(* IEC 61131-3 sources: TA/Tests/RetainTest/OLD/Structure test (part 8) *)

    ARRAY_ARRAY_STRUCTURE_AUTO.ARRAY_ARRAY_SINT[3][0] := ARRAY_ARRAY_STRUCTURE_AUTO.ARRAY_ARRAY_SINT[3][0] + 1;
    ARRAY_ARRAY_STRUCTURE_AUTO.ARRAY_ARRAY_SINT[3][1] := ARRAY_ARRAY_STRUCTURE_AUTO.ARRAY_ARRAY_SINT[3][1] + 1;
    ARRAY_ARRAY_STRUCTURE_AUTO.ARRAY_ARRAY_SINT[3][2] := ARRAY_ARRAY_STRUCTURE_AUTO.ARRAY_ARRAY_SINT[3][2] + 1;
    ARRAY_ARRAY_STRUCTURE_AUTO.ARRAY_ARRAY_SINT[3][3] := ARRAY_ARRAY_STRUCTURE_AUTO.ARRAY_ARRAY_SINT[3][3] + 1;
    ARRAY_ARRAY_STRUCTURE_AUTO.ARRAY_ARRAY_SINT[3][4] := ARRAY_ARRAY_STRUCTURE_AUTO.ARRAY_ARRAY_SINT[3][4] + 1;
    ARRAY_ARRAY_STRUCTURE_AUTO.ARRAY_ARRAY_SINT[3][5] := ARRAY_ARRAY_STRUCTURE_AUTO.ARRAY_ARRAY_SINT[3][5] + 1;
    ARRAY_ARRAY_STRUCTURE_AUTO.ARRAY_ARRAY_SINT[3][6] := ARRAY_ARRAY_STRUCTURE_AUTO.ARRAY_ARRAY_SINT[3][6] + 1;
    ARRAY_ARRAY_STRUCTURE_AUTO.ARRAY_ARRAY_SINT[3][7] := ARRAY_ARRAY_STRUCTURE_AUTO.ARRAY_ARRAY_SINT[3][7] + 1;
    ARRAY_ARRAY_STRUCTURE_AUTO.ARRAY_ARRAY_SINT[3][8] := ARRAY_ARRAY_STRUCTURE_AUTO.ARRAY_ARRAY_SINT[3][8] + 1;
    ARRAY_ARRAY_STRUCTURE_AUTO.ARRAY_ARRAY_SINT[3][9] := ARRAY_ARRAY_STRUCTURE_AUTO.ARRAY_ARRAY_SINT[3][9] + 1;

    ARRAY_ARRAY_STRUCTURE_AUTO.ARRAY_ARRAY_SINT[4][0] := ARRAY_ARRAY_STRUCTURE_AUTO.ARRAY_ARRAY_SINT[4][0] + 1;
    ARRAY_ARRAY_STRUCTURE_AUTO.ARRAY_ARRAY_SINT[4][1] := ARRAY_ARRAY_STRUCTURE_AUTO.ARRAY_ARRAY_SINT[4][1] + 1;
    ARRAY_ARRAY_STRUCTURE_AUTO.ARRAY_ARRAY_SINT[4][2] := ARRAY_ARRAY_STRUCTURE_AUTO.ARRAY_ARRAY_SINT[4][2] + 1;
    ARRAY_ARRAY_STRUCTURE_AUTO.ARRAY_ARRAY_SINT[4][3] := ARRAY_ARRAY_STRUCTURE_AUTO.ARRAY_ARRAY_SINT[4][3] + 1;
    ARRAY_ARRAY_STRUCTURE_AUTO.ARRAY_ARRAY_SINT[4][4] := ARRAY_ARRAY_STRUCTURE_AUTO.ARRAY_ARRAY_SINT[4][4] + 1;
    ARRAY_ARRAY_STRUCTURE_AUTO.ARRAY_ARRAY_SINT[4][5] := ARRAY_ARRAY_STRUCTURE_AUTO.ARRAY_ARRAY_SINT[4][5] + 1;
    ARRAY_ARRAY_STRUCTURE_AUTO.ARRAY_ARRAY_SINT[4][6] := ARRAY_ARRAY_STRUCTURE_AUTO.ARRAY_ARRAY_SINT[4][6] + 1;
    ARRAY_ARRAY_STRUCTURE_AUTO.ARRAY_ARRAY_SINT[4][7] := ARRAY_ARRAY_STRUCTURE_AUTO.ARRAY_ARRAY_SINT[4][7] + 1;
    ARRAY_ARRAY_STRUCTURE_AUTO.ARRAY_ARRAY_SINT[4][8] := ARRAY_ARRAY_STRUCTURE_AUTO.ARRAY_ARRAY_SINT[4][8] + 1;
    ARRAY_ARRAY_STRUCTURE_AUTO.ARRAY_ARRAY_SINT[4][9] := ARRAY_ARRAY_STRUCTURE_AUTO.ARRAY_ARRAY_SINT[4][9] + 1;

    ARRAY_ARRAY_STRUCTURE_AUTO.ARRAY_ARRAY_SINT[5][0] := ARRAY_ARRAY_STRUCTURE_AUTO.ARRAY_ARRAY_SINT[5][0] + 1;
    ARRAY_ARRAY_STRUCTURE_AUTO.ARRAY_ARRAY_SINT[5][1] := ARRAY_ARRAY_STRUCTURE_AUTO.ARRAY_ARRAY_SINT[5][1] + 1;
    ARRAY_ARRAY_STRUCTURE_AUTO.ARRAY_ARRAY_SINT[5][2] := ARRAY_ARRAY_STRUCTURE_AUTO.ARRAY_ARRAY_SINT[5][2] + 1;
    ARRAY_ARRAY_STRUCTURE_AUTO.ARRAY_ARRAY_SINT[5][3] := ARRAY_ARRAY_STRUCTURE_AUTO.ARRAY_ARRAY_SINT[5][3] + 1;
    ARRAY_ARRAY_STRUCTURE_AUTO.ARRAY_ARRAY_SINT[5][4] := ARRAY_ARRAY_STRUCTURE_AUTO.ARRAY_ARRAY_SINT[5][4] + 1;
    ARRAY_ARRAY_STRUCTURE_AUTO.ARRAY_ARRAY_SINT[5][5] := ARRAY_ARRAY_STRUCTURE_AUTO.ARRAY_ARRAY_SINT[5][5] + 1;
    ARRAY_ARRAY_STRUCTURE_AUTO.ARRAY_ARRAY_SINT[5][6] := ARRAY_ARRAY_STRUCTURE_AUTO.ARRAY_ARRAY_SINT[5][6] + 1;
    ARRAY_ARRAY_STRUCTURE_AUTO.ARRAY_ARRAY_SINT[5][7] := ARRAY_ARRAY_STRUCTURE_AUTO.ARRAY_ARRAY_SINT[5][7] + 1;
    ARRAY_ARRAY_STRUCTURE_AUTO.ARRAY_ARRAY_SINT[5][8] := ARRAY_ARRAY_STRUCTURE_AUTO.ARRAY_ARRAY_SINT[5][8] + 1;
    ARRAY_ARRAY_STRUCTURE_AUTO.ARRAY_ARRAY_SINT[5][9] := ARRAY_ARRAY_STRUCTURE_AUTO.ARRAY_ARRAY_SINT[5][9] + 1;

    ARRAY_ARRAY_STRUCTURE_AUTO.ARRAY_ARRAY_SINT[6][0] := ARRAY_ARRAY_STRUCTURE_AUTO.ARRAY_ARRAY_SINT[6][0] + 1;
    ARRAY_ARRAY_STRUCTURE_AUTO.ARRAY_ARRAY_SINT[6][1] := ARRAY_ARRAY_STRUCTURE_AUTO.ARRAY_ARRAY_SINT[6][1] + 1;
    ARRAY_ARRAY_STRUCTURE_AUTO.ARRAY_ARRAY_SINT[6][2] := ARRAY_ARRAY_STRUCTURE_AUTO.ARRAY_ARRAY_SINT[6][2] + 1;
    ARRAY_ARRAY_STRUCTURE_AUTO.ARRAY_ARRAY_SINT[6][3] := ARRAY_ARRAY_STRUCTURE_AUTO.ARRAY_ARRAY_SINT[6][3] + 1;
    ARRAY_ARRAY_STRUCTURE_AUTO.ARRAY_ARRAY_SINT[6][4] := ARRAY_ARRAY_STRUCTURE_AUTO.ARRAY_ARRAY_SINT[6][4] + 1;
    ARRAY_ARRAY_STRUCTURE_AUTO.ARRAY_ARRAY_SINT[6][5] := ARRAY_ARRAY_STRUCTURE_AUTO.ARRAY_ARRAY_SINT[6][5] + 1;
    ARRAY_ARRAY_STRUCTURE_AUTO.ARRAY_ARRAY_SINT[6][6] := ARRAY_ARRAY_STRUCTURE_AUTO.ARRAY_ARRAY_SINT[6][6] + 1;
    ARRAY_ARRAY_STRUCTURE_AUTO.ARRAY_ARRAY_SINT[6][7] := ARRAY_ARRAY_STRUCTURE_AUTO.ARRAY_ARRAY_SINT[6][7] + 1;
    ARRAY_ARRAY_STRUCTURE_AUTO.ARRAY_ARRAY_SINT[6][8] := ARRAY_ARRAY_STRUCTURE_AUTO.ARRAY_ARRAY_SINT[6][8] + 1;
    ARRAY_ARRAY_STRUCTURE_AUTO.ARRAY_ARRAY_SINT[6][9] := ARRAY_ARRAY_STRUCTURE_AUTO.ARRAY_ARRAY_SINT[6][9] + 1;

    ARRAY_ARRAY_STRUCTURE_AUTO.ARRAY_ARRAY_SINT[7][0] := ARRAY_ARRAY_STRUCTURE_AUTO.ARRAY_ARRAY_SINT[6][0];
    ARRAY_ARRAY_STRUCTURE_AUTO.ARRAY_ARRAY_SINT[7][1] := ARRAY_ARRAY_STRUCTURE_AUTO.ARRAY_ARRAY_SINT[6][1];
    ARRAY_ARRAY_STRUCTURE_AUTO.ARRAY_ARRAY_SINT[7][2] := ARRAY_ARRAY_STRUCTURE_AUTO.ARRAY_ARRAY_SINT[6][2];
    ARRAY_ARRAY_STRUCTURE_AUTO.ARRAY_ARRAY_SINT[7][3] := ARRAY_ARRAY_STRUCTURE_AUTO.ARRAY_ARRAY_SINT[6][3];
    ARRAY_ARRAY_STRUCTURE_AUTO.ARRAY_ARRAY_SINT[7][4] := ARRAY_ARRAY_STRUCTURE_AUTO.ARRAY_ARRAY_SINT[6][4];
    ARRAY_ARRAY_STRUCTURE_AUTO.ARRAY_ARRAY_SINT[7][5] := ARRAY_ARRAY_STRUCTURE_AUTO.ARRAY_ARRAY_SINT[6][5];
    ARRAY_ARRAY_STRUCTURE_AUTO.ARRAY_ARRAY_SINT[7][6] := ARRAY_ARRAY_STRUCTURE_AUTO.ARRAY_ARRAY_SINT[6][6];
    ARRAY_ARRAY_STRUCTURE_AUTO.ARRAY_ARRAY_SINT[7][7] := ARRAY_ARRAY_STRUCTURE_AUTO.ARRAY_ARRAY_SINT[6][7];
    ARRAY_ARRAY_STRUCTURE_AUTO.ARRAY_ARRAY_SINT[7][8] := ARRAY_ARRAY_STRUCTURE_AUTO.ARRAY_ARRAY_SINT[6][8];
    ARRAY_ARRAY_STRUCTURE_AUTO.ARRAY_ARRAY_SINT[7][9] := ARRAY_ARRAY_STRUCTURE_AUTO.ARRAY_ARRAY_SINT[6][9];

    ARRAY_ARRAY_STRUCTURE_AUTO.ARRAY_ARRAY_STRING[0][0] := ANY_TO_STRING(ARRAY_ARRAY_STRUCTURE_AUTO.ARRAY_ARRAY_DINT[0][0]) + ' ' + ANY_TO_STRING(ARRAY_ARRAY_STRUCTURE_AUTO.ARRAY_ARRAY_TIME[0][0]);
    ARRAY_ARRAY_STRUCTURE_AUTO.ARRAY_ARRAY_STRING[0][1] := ANY_TO_STRING(ARRAY_ARRAY_STRUCTURE_AUTO.ARRAY_ARRAY_DINT[0][1]) + ' ' + ANY_TO_STRING(ARRAY_ARRAY_STRUCTURE_AUTO.ARRAY_ARRAY_TIME[0][1]);
    ARRAY_ARRAY_STRUCTURE_AUTO.ARRAY_ARRAY_STRING[0][2] := ANY_TO_STRING(ARRAY_ARRAY_STRUCTURE_AUTO.ARRAY_ARRAY_DINT[0][2]) + ' ' + ANY_TO_STRING(ARRAY_ARRAY_STRUCTURE_AUTO.ARRAY_ARRAY_TIME[0][2]);
    ARRAY_ARRAY_STRUCTURE_AUTO.ARRAY_ARRAY_STRING[0][3] := ANY_TO_STRING(ARRAY_ARRAY_STRUCTURE_AUTO.ARRAY_ARRAY_DINT[0][3]) + ' ' + ANY_TO_STRING(ARRAY_ARRAY_STRUCTURE_AUTO.ARRAY_ARRAY_TIME[0][3]);
    ARRAY_ARRAY_STRUCTURE_AUTO.ARRAY_ARRAY_STRING[0][4] := ANY_TO_STRING(ARRAY_ARRAY_STRUCTURE_AUTO.ARRAY_ARRAY_DINT[0][4]) + ' ' + ANY_TO_STRING(ARRAY_ARRAY_STRUCTURE_AUTO.ARRAY_ARRAY_TIME[0][4]);
    ARRAY_ARRAY_STRUCTURE_AUTO.ARRAY_ARRAY_STRING[0][5] := ANY_TO_STRING(ARRAY_ARRAY_STRUCTURE_AUTO.ARRAY_ARRAY_DINT[0][5]) + ' ' + ANY_TO_STRING(ARRAY_ARRAY_STRUCTURE_AUTO.ARRAY_ARRAY_TIME[0][5]);
    ARRAY_ARRAY_STRUCTURE_AUTO.ARRAY_ARRAY_STRING[0][6] := ANY_TO_STRING(ARRAY_ARRAY_STRUCTURE_AUTO.ARRAY_ARRAY_DINT[0][6]) + ' ' + ANY_TO_STRING(ARRAY_ARRAY_STRUCTURE_AUTO.ARRAY_ARRAY_TIME[0][6]);
    ARRAY_ARRAY_STRUCTURE_AUTO.ARRAY_ARRAY_STRING[0][7] := ANY_TO_STRING(ARRAY_ARRAY_STRUCTURE_AUTO.ARRAY_ARRAY_DINT[0][7]) + ' ' + ANY_TO_STRING(ARRAY_ARRAY_STRUCTURE_AUTO.ARRAY_ARRAY_TIME[0][7]);
    ARRAY_ARRAY_STRUCTURE_AUTO.ARRAY_ARRAY_STRING[0][8] := ARRAY_ARRAY_STRUCTURE_AUTO.ARRAY_ARRAY_STRING[0][6];
    ARRAY_ARRAY_STRUCTURE_AUTO.ARRAY_ARRAY_STRING[0][9] := ARRAY_ARRAY_STRUCTURE_AUTO.ARRAY_ARRAY_STRING[0][7];

    ARRAY_ARRAY_STRUCTURE_AUTO.ARRAY_ARRAY_STRING[1][0] := ANY_TO_STRING(ARRAY_ARRAY_STRUCTURE_AUTO.ARRAY_ARRAY_DINT[1][0]) + ' ' + ANY_TO_STRING(ARRAY_ARRAY_STRUCTURE_AUTO.ARRAY_ARRAY_TIME[1][0]);
    ARRAY_ARRAY_STRUCTURE_AUTO.ARRAY_ARRAY_STRING[1][1] := ANY_TO_STRING(ARRAY_ARRAY_STRUCTURE_AUTO.ARRAY_ARRAY_DINT[1][1]) + ' ' + ANY_TO_STRING(ARRAY_ARRAY_STRUCTURE_AUTO.ARRAY_ARRAY_TIME[1][1]);
    ARRAY_ARRAY_STRUCTURE_AUTO.ARRAY_ARRAY_STRING[1][2] := ANY_TO_STRING(ARRAY_ARRAY_STRUCTURE_AUTO.ARRAY_ARRAY_DINT[1][2]) + ' ' + ANY_TO_STRING(ARRAY_ARRAY_STRUCTURE_AUTO.ARRAY_ARRAY_TIME[1][2]);
    ARRAY_ARRAY_STRUCTURE_AUTO.ARRAY_ARRAY_STRING[1][3] := ANY_TO_STRING(ARRAY_ARRAY_STRUCTURE_AUTO.ARRAY_ARRAY_DINT[1][3]) + ' ' + ANY_TO_STRING(ARRAY_ARRAY_STRUCTURE_AUTO.ARRAY_ARRAY_TIME[1][3]);
    ARRAY_ARRAY_STRUCTURE_AUTO.ARRAY_ARRAY_STRING[1][4] := ANY_TO_STRING(ARRAY_ARRAY_STRUCTURE_AUTO.ARRAY_ARRAY_DINT[1][4]) + ' ' + ANY_TO_STRING(ARRAY_ARRAY_STRUCTURE_AUTO.ARRAY_ARRAY_TIME[1][4]);
    ARRAY_ARRAY_STRUCTURE_AUTO.ARRAY_ARRAY_STRING[1][5] := ANY_TO_STRING(ARRAY_ARRAY_STRUCTURE_AUTO.ARRAY_ARRAY_DINT[1][5]) + ' ' + ANY_TO_STRING(ARRAY_ARRAY_STRUCTURE_AUTO.ARRAY_ARRAY_TIME[1][5]);
    ARRAY_ARRAY_STRUCTURE_AUTO.ARRAY_ARRAY_STRING[1][6] := ANY_TO_STRING(ARRAY_ARRAY_STRUCTURE_AUTO.ARRAY_ARRAY_DINT[1][6]) + ' ' + ANY_TO_STRING(ARRAY_ARRAY_STRUCTURE_AUTO.ARRAY_ARRAY_TIME[1][6]);
    ARRAY_ARRAY_STRUCTURE_AUTO.ARRAY_ARRAY_STRING[1][7] := ANY_TO_STRING(ARRAY_ARRAY_STRUCTURE_AUTO.ARRAY_ARRAY_DINT[1][7]) + ' ' + ANY_TO_STRING(ARRAY_ARRAY_STRUCTURE_AUTO.ARRAY_ARRAY_TIME[1][7]);
    ARRAY_ARRAY_STRUCTURE_AUTO.ARRAY_ARRAY_STRING[1][8] := ARRAY_ARRAY_STRUCTURE_AUTO.ARRAY_ARRAY_STRING[1][6];
    ARRAY_ARRAY_STRUCTURE_AUTO.ARRAY_ARRAY_STRING[1][9] := ARRAY_ARRAY_STRUCTURE_AUTO.ARRAY_ARRAY_STRING[1][7];

    ARRAY_ARRAY_STRUCTURE_AUTO.ARRAY_ARRAY_STRING[2][0] := ANY_TO_STRING(ARRAY_ARRAY_STRUCTURE_AUTO.ARRAY_ARRAY_DINT[2][0]) + ' ' + ANY_TO_STRING(ARRAY_ARRAY_STRUCTURE_AUTO.ARRAY_ARRAY_TIME[2][0]);
    ARRAY_ARRAY_STRUCTURE_AUTO.ARRAY_ARRAY_STRING[2][1] := ANY_TO_STRING(ARRAY_ARRAY_STRUCTURE_AUTO.ARRAY_ARRAY_DINT[2][1]) + ' ' + ANY_TO_STRING(ARRAY_ARRAY_STRUCTURE_AUTO.ARRAY_ARRAY_TIME[2][1]);
    ARRAY_ARRAY_STRUCTURE_AUTO.ARRAY_ARRAY_STRING[2][2] := ANY_TO_STRING(ARRAY_ARRAY_STRUCTURE_AUTO.ARRAY_ARRAY_DINT[2][2]) + ' ' + ANY_TO_STRING(ARRAY_ARRAY_STRUCTURE_AUTO.ARRAY_ARRAY_TIME[2][2]);
    ARRAY_ARRAY_STRUCTURE_AUTO.ARRAY_ARRAY_STRING[2][3] := ANY_TO_STRING(ARRAY_ARRAY_STRUCTURE_AUTO.ARRAY_ARRAY_DINT[2][3]) + ' ' + ANY_TO_STRING(ARRAY_ARRAY_STRUCTURE_AUTO.ARRAY_ARRAY_TIME[2][3]);
    ARRAY_ARRAY_STRUCTURE_AUTO.ARRAY_ARRAY_STRING[2][4] := ANY_TO_STRING(ARRAY_ARRAY_STRUCTURE_AUTO.ARRAY_ARRAY_DINT[2][4]) + ' ' + ANY_TO_STRING(ARRAY_ARRAY_STRUCTURE_AUTO.ARRAY_ARRAY_TIME[2][4]);
    ARRAY_ARRAY_STRUCTURE_AUTO.ARRAY_ARRAY_STRING[2][5] := ANY_TO_STRING(ARRAY_ARRAY_STRUCTURE_AUTO.ARRAY_ARRAY_DINT[2][5]) + ' ' + ANY_TO_STRING(ARRAY_ARRAY_STRUCTURE_AUTO.ARRAY_ARRAY_TIME[2][5]);
    ARRAY_ARRAY_STRUCTURE_AUTO.ARRAY_ARRAY_STRING[2][6] := ANY_TO_STRING(ARRAY_ARRAY_STRUCTURE_AUTO.ARRAY_ARRAY_DINT[2][6]) + ' ' + ANY_TO_STRING(ARRAY_ARRAY_STRUCTURE_AUTO.ARRAY_ARRAY_TIME[2][6]);
    ARRAY_ARRAY_STRUCTURE_AUTO.ARRAY_ARRAY_STRING[2][7] := ANY_TO_STRING(ARRAY_ARRAY_STRUCTURE_AUTO.ARRAY_ARRAY_DINT[2][7]) + ' ' + ANY_TO_STRING(ARRAY_ARRAY_STRUCTURE_AUTO.ARRAY_ARRAY_TIME[2][7]);
    ARRAY_ARRAY_STRUCTURE_AUTO.ARRAY_ARRAY_STRING[2][8] := ANY_TO_STRING(ARRAY_ARRAY_STRUCTURE_AUTO.ARRAY_ARRAY_DINT[2][8]) + ' ' + ANY_TO_STRING(ARRAY_ARRAY_STRUCTURE_AUTO.ARRAY_ARRAY_TIME[2][8]);
    ARRAY_ARRAY_STRUCTURE_AUTO.ARRAY_ARRAY_STRING[2][9] := ANY_TO_STRING(ARRAY_ARRAY_STRUCTURE_AUTO.ARRAY_ARRAY_DINT[2][9]) + ' ' + ANY_TO_STRING(ARRAY_ARRAY_STRUCTURE_AUTO.ARRAY_ARRAY_TIME[2][9]);

    ARRAY_ARRAY_STRUCTURE_AUTO.ARRAY_ARRAY_STRING[3][0] := ANY_TO_STRING(ARRAY_ARRAY_STRUCTURE_AUTO.ARRAY_ARRAY_DINT[3][0]) + ' ' + ANY_TO_STRING(ARRAY_ARRAY_STRUCTURE_AUTO.ARRAY_ARRAY_TIME[3][0]);
    ARRAY_ARRAY_STRUCTURE_AUTO.ARRAY_ARRAY_STRING[3][1] := ANY_TO_STRING(ARRAY_ARRAY_STRUCTURE_AUTO.ARRAY_ARRAY_DINT[3][1]) + ' ' + ANY_TO_STRING(ARRAY_ARRAY_STRUCTURE_AUTO.ARRAY_ARRAY_TIME[3][1]);
    ARRAY_ARRAY_STRUCTURE_AUTO.ARRAY_ARRAY_STRING[3][2] := ANY_TO_STRING(ARRAY_ARRAY_STRUCTURE_AUTO.ARRAY_ARRAY_DINT[3][2]) + ' ' + ANY_TO_STRING(ARRAY_ARRAY_STRUCTURE_AUTO.ARRAY_ARRAY_TIME[3][2]);
    ARRAY_ARRAY_STRUCTURE_AUTO.ARRAY_ARRAY_STRING[3][3] := ANY_TO_STRING(ARRAY_ARRAY_STRUCTURE_AUTO.ARRAY_ARRAY_DINT[3][3]) + ' ' + ANY_TO_STRING(ARRAY_ARRAY_STRUCTURE_AUTO.ARRAY_ARRAY_TIME[3][3]);
    ARRAY_ARRAY_STRUCTURE_AUTO.ARRAY_ARRAY_STRING[3][4] := ANY_TO_STRING(ARRAY_ARRAY_STRUCTURE_AUTO.ARRAY_ARRAY_DINT[3][4]) + ' ' + ANY_TO_STRING(ARRAY_ARRAY_STRUCTURE_AUTO.ARRAY_ARRAY_TIME[3][4]);
    ARRAY_ARRAY_STRUCTURE_AUTO.ARRAY_ARRAY_STRING[3][5] := ANY_TO_STRING(ARRAY_ARRAY_STRUCTURE_AUTO.ARRAY_ARRAY_DINT[3][5]) + ' ' + ANY_TO_STRING(ARRAY_ARRAY_STRUCTURE_AUTO.ARRAY_ARRAY_TIME[3][5]);
    ARRAY_ARRAY_STRUCTURE_AUTO.ARRAY_ARRAY_STRING[3][6] := ANY_TO_STRING(ARRAY_ARRAY_STRUCTURE_AUTO.ARRAY_ARRAY_DINT[3][6]) + ' ' + ANY_TO_STRING(ARRAY_ARRAY_STRUCTURE_AUTO.ARRAY_ARRAY_TIME[3][6]);
    ARRAY_ARRAY_STRUCTURE_AUTO.ARRAY_ARRAY_STRING[3][7] := ANY_TO_STRING(ARRAY_ARRAY_STRUCTURE_AUTO.ARRAY_ARRAY_DINT[3][7]) + ' ' + ANY_TO_STRING(ARRAY_ARRAY_STRUCTURE_AUTO.ARRAY_ARRAY_TIME[3][7]);
    ARRAY_ARRAY_STRUCTURE_AUTO.ARRAY_ARRAY_STRING[3][8] := ANY_TO_STRING(ARRAY_ARRAY_STRUCTURE_AUTO.ARRAY_ARRAY_DINT[3][8]) + ' ' + ANY_TO_STRING(ARRAY_ARRAY_STRUCTURE_AUTO.ARRAY_ARRAY_TIME[3][8]);
    ARRAY_ARRAY_STRUCTURE_AUTO.ARRAY_ARRAY_STRING[3][9] := ANY_TO_STRING(ARRAY_ARRAY_STRUCTURE_AUTO.ARRAY_ARRAY_DINT[3][9]) + ' ' + ANY_TO_STRING(ARRAY_ARRAY_STRUCTURE_AUTO.ARRAY_ARRAY_TIME[3][9]);

    ARRAY_ARRAY_STRUCTURE_AUTO.ARRAY_ARRAY_STRING[4][0] := ANY_TO_STRING(ARRAY_ARRAY_STRUCTURE_AUTO.ARRAY_ARRAY_DINT[4][0]) + ' ' + ANY_TO_STRING(ARRAY_ARRAY_STRUCTURE_AUTO.ARRAY_ARRAY_TIME[4][0]);
    ARRAY_ARRAY_STRUCTURE_AUTO.ARRAY_ARRAY_STRING[4][1] := ANY_TO_STRING(ARRAY_ARRAY_STRUCTURE_AUTO.ARRAY_ARRAY_DINT[4][1]) + ' ' + ANY_TO_STRING(ARRAY_ARRAY_STRUCTURE_AUTO.ARRAY_ARRAY_TIME[4][1]);
    ARRAY_ARRAY_STRUCTURE_AUTO.ARRAY_ARRAY_STRING[4][2] := ANY_TO_STRING(ARRAY_ARRAY_STRUCTURE_AUTO.ARRAY_ARRAY_DINT[4][2]) + ' ' + ANY_TO_STRING(ARRAY_ARRAY_STRUCTURE_AUTO.ARRAY_ARRAY_TIME[4][2]);
    ARRAY_ARRAY_STRUCTURE_AUTO.ARRAY_ARRAY_STRING[4][3] := ANY_TO_STRING(ARRAY_ARRAY_STRUCTURE_AUTO.ARRAY_ARRAY_DINT[4][3]) + ' ' + ANY_TO_STRING(ARRAY_ARRAY_STRUCTURE_AUTO.ARRAY_ARRAY_TIME[4][3]);
    ARRAY_ARRAY_STRUCTURE_AUTO.ARRAY_ARRAY_STRING[4][4] := ANY_TO_STRING(ARRAY_ARRAY_STRUCTURE_AUTO.ARRAY_ARRAY_DINT[4][4]) + ' ' + ANY_TO_STRING(ARRAY_ARRAY_STRUCTURE_AUTO.ARRAY_ARRAY_TIME[4][4]);
    ARRAY_ARRAY_STRUCTURE_AUTO.ARRAY_ARRAY_STRING[4][5] := ANY_TO_STRING(ARRAY_ARRAY_STRUCTURE_AUTO.ARRAY_ARRAY_DINT[4][5]) + ' ' + ANY_TO_STRING(ARRAY_ARRAY_STRUCTURE_AUTO.ARRAY_ARRAY_TIME[4][5]);
    ARRAY_ARRAY_STRUCTURE_AUTO.ARRAY_ARRAY_STRING[4][6] := ANY_TO_STRING(ARRAY_ARRAY_STRUCTURE_AUTO.ARRAY_ARRAY_DINT[4][6]) + ' ' + ANY_TO_STRING(ARRAY_ARRAY_STRUCTURE_AUTO.ARRAY_ARRAY_TIME[4][6]);
    ARRAY_ARRAY_STRUCTURE_AUTO.ARRAY_ARRAY_STRING[4][7] := ANY_TO_STRING(ARRAY_ARRAY_STRUCTURE_AUTO.ARRAY_ARRAY_DINT[4][7]) + ' ' + ANY_TO_STRING(ARRAY_ARRAY_STRUCTURE_AUTO.ARRAY_ARRAY_TIME[4][7]);
    ARRAY_ARRAY_STRUCTURE_AUTO.ARRAY_ARRAY_STRING[4][8] := ANY_TO_STRING(ARRAY_ARRAY_STRUCTURE_AUTO.ARRAY_ARRAY_DINT[4][8]) + ' ' + ANY_TO_STRING(ARRAY_ARRAY_STRUCTURE_AUTO.ARRAY_ARRAY_TIME[4][8]);
    ARRAY_ARRAY_STRUCTURE_AUTO.ARRAY_ARRAY_STRING[4][9] := ANY_TO_STRING(ARRAY_ARRAY_STRUCTURE_AUTO.ARRAY_ARRAY_DINT[4][9]) + ' ' + ANY_TO_STRING(ARRAY_ARRAY_STRUCTURE_AUTO.ARRAY_ARRAY_TIME[4][9]);

    ARRAY_ARRAY_STRUCTURE_AUTO.ARRAY_ARRAY_STRING[5][0] := ANY_TO_STRING(ARRAY_ARRAY_STRUCTURE_AUTO.ARRAY_ARRAY_DINT[5][0]) + ' ' + ANY_TO_STRING(ARRAY_ARRAY_STRUCTURE_AUTO.ARRAY_ARRAY_TIME[5][0]);
    ARRAY_ARRAY_STRUCTURE_AUTO.ARRAY_ARRAY_STRING[5][1] := ANY_TO_STRING(ARRAY_ARRAY_STRUCTURE_AUTO.ARRAY_ARRAY_DINT[5][1]) + ' ' + ANY_TO_STRING(ARRAY_ARRAY_STRUCTURE_AUTO.ARRAY_ARRAY_TIME[5][1]);
    ARRAY_ARRAY_STRUCTURE_AUTO.ARRAY_ARRAY_STRING[5][2] := ANY_TO_STRING(ARRAY_ARRAY_STRUCTURE_AUTO.ARRAY_ARRAY_DINT[5][2]) + ' ' + ANY_TO_STRING(ARRAY_ARRAY_STRUCTURE_AUTO.ARRAY_ARRAY_TIME[5][2]);
    ARRAY_ARRAY_STRUCTURE_AUTO.ARRAY_ARRAY_STRING[5][3] := ANY_TO_STRING(ARRAY_ARRAY_STRUCTURE_AUTO.ARRAY_ARRAY_DINT[5][3]) + ' ' + ANY_TO_STRING(ARRAY_ARRAY_STRUCTURE_AUTO.ARRAY_ARRAY_TIME[5][3]);
    ARRAY_ARRAY_STRUCTURE_AUTO.ARRAY_ARRAY_STRING[5][4] := ANY_TO_STRING(ARRAY_ARRAY_STRUCTURE_AUTO.ARRAY_ARRAY_DINT[5][4]) + ' ' + ANY_TO_STRING(ARRAY_ARRAY_STRUCTURE_AUTO.ARRAY_ARRAY_TIME[5][4]);
    ARRAY_ARRAY_STRUCTURE_AUTO.ARRAY_ARRAY_STRING[5][5] := ANY_TO_STRING(ARRAY_ARRAY_STRUCTURE_AUTO.ARRAY_ARRAY_DINT[5][5]) + ' ' + ANY_TO_STRING(ARRAY_ARRAY_STRUCTURE_AUTO.ARRAY_ARRAY_TIME[5][5]);
    ARRAY_ARRAY_STRUCTURE_AUTO.ARRAY_ARRAY_STRING[5][6] := ANY_TO_STRING(ARRAY_ARRAY_STRUCTURE_AUTO.ARRAY_ARRAY_DINT[5][6]) + ' ' + ANY_TO_STRING(ARRAY_ARRAY_STRUCTURE_AUTO.ARRAY_ARRAY_TIME[5][6]);
    ARRAY_ARRAY_STRUCTURE_AUTO.ARRAY_ARRAY_STRING[5][7] := ANY_TO_STRING(ARRAY_ARRAY_STRUCTURE_AUTO.ARRAY_ARRAY_DINT[5][7]) + ' ' + ANY_TO_STRING(ARRAY_ARRAY_STRUCTURE_AUTO.ARRAY_ARRAY_TIME[5][7]);
    ARRAY_ARRAY_STRUCTURE_AUTO.ARRAY_ARRAY_STRING[5][8] := ANY_TO_STRING(ARRAY_ARRAY_STRUCTURE_AUTO.ARRAY_ARRAY_DINT[5][8]) + ' ' + ANY_TO_STRING(ARRAY_ARRAY_STRUCTURE_AUTO.ARRAY_ARRAY_TIME[5][8]);
    ARRAY_ARRAY_STRUCTURE_AUTO.ARRAY_ARRAY_STRING[5][9] := ANY_TO_STRING(ARRAY_ARRAY_STRUCTURE_AUTO.ARRAY_ARRAY_DINT[5][9]) + ' ' + ANY_TO_STRING(ARRAY_ARRAY_STRUCTURE_AUTO.ARRAY_ARRAY_TIME[5][9]);

    ARRAY_ARRAY_STRUCTURE_AUTO.ARRAY_ARRAY_STRING[6][0] := ANY_TO_STRING(ARRAY_ARRAY_STRUCTURE_AUTO.ARRAY_ARRAY_DINT[6][0]) + ' ' + ANY_TO_STRING(ARRAY_ARRAY_STRUCTURE_AUTO.ARRAY_ARRAY_TIME[6][0]);
    ARRAY_ARRAY_STRUCTURE_AUTO.ARRAY_ARRAY_STRING[6][1] := ANY_TO_STRING(ARRAY_ARRAY_STRUCTURE_AUTO.ARRAY_ARRAY_DINT[6][1]) + ' ' + ANY_TO_STRING(ARRAY_ARRAY_STRUCTURE_AUTO.ARRAY_ARRAY_TIME[6][1]);
    ARRAY_ARRAY_STRUCTURE_AUTO.ARRAY_ARRAY_STRING[6][2] := ANY_TO_STRING(ARRAY_ARRAY_STRUCTURE_AUTO.ARRAY_ARRAY_DINT[6][2]) + ' ' + ANY_TO_STRING(ARRAY_ARRAY_STRUCTURE_AUTO.ARRAY_ARRAY_TIME[6][2]);
    ARRAY_ARRAY_STRUCTURE_AUTO.ARRAY_ARRAY_STRING[6][3] := ANY_TO_STRING(ARRAY_ARRAY_STRUCTURE_AUTO.ARRAY_ARRAY_DINT[6][3]) + ' ' + ANY_TO_STRING(ARRAY_ARRAY_STRUCTURE_AUTO.ARRAY_ARRAY_TIME[6][3]);
    ARRAY_ARRAY_STRUCTURE_AUTO.ARRAY_ARRAY_STRING[6][4] := ANY_TO_STRING(ARRAY_ARRAY_STRUCTURE_AUTO.ARRAY_ARRAY_DINT[6][4]) + ' ' + ANY_TO_STRING(ARRAY_ARRAY_STRUCTURE_AUTO.ARRAY_ARRAY_TIME[6][4]);
    ARRAY_ARRAY_STRUCTURE_AUTO.ARRAY_ARRAY_STRING[6][5] := ANY_TO_STRING(ARRAY_ARRAY_STRUCTURE_AUTO.ARRAY_ARRAY_DINT[6][5]) + ' ' + ANY_TO_STRING(ARRAY_ARRAY_STRUCTURE_AUTO.ARRAY_ARRAY_TIME[6][5]);
    ARRAY_ARRAY_STRUCTURE_AUTO.ARRAY_ARRAY_STRING[6][6] := ANY_TO_STRING(ARRAY_ARRAY_STRUCTURE_AUTO.ARRAY_ARRAY_DINT[6][6]) + ' ' + ANY_TO_STRING(ARRAY_ARRAY_STRUCTURE_AUTO.ARRAY_ARRAY_TIME[6][6]);
    ARRAY_ARRAY_STRUCTURE_AUTO.ARRAY_ARRAY_STRING[6][7] := ANY_TO_STRING(ARRAY_ARRAY_STRUCTURE_AUTO.ARRAY_ARRAY_DINT[6][7]) + ' ' + ANY_TO_STRING(ARRAY_ARRAY_STRUCTURE_AUTO.ARRAY_ARRAY_TIME[6][7]);
    ARRAY_ARRAY_STRUCTURE_AUTO.ARRAY_ARRAY_STRING[6][8] := ANY_TO_STRING(ARRAY_ARRAY_STRUCTURE_AUTO.ARRAY_ARRAY_DINT[6][8]) + ' ' + ANY_TO_STRING(ARRAY_ARRAY_STRUCTURE_AUTO.ARRAY_ARRAY_TIME[6][8]);
    ARRAY_ARRAY_STRUCTURE_AUTO.ARRAY_ARRAY_STRING[6][9] := ANY_TO_STRING(ARRAY_ARRAY_STRUCTURE_AUTO.ARRAY_ARRAY_DINT[6][9]) + ' ' + ANY_TO_STRING(ARRAY_ARRAY_STRUCTURE_AUTO.ARRAY_ARRAY_TIME[6][9]);

    ARRAY_ARRAY_STRUCTURE_AUTO.ARRAY_ARRAY_STRING[7][0] := ARRAY_ARRAY_STRUCTURE_AUTO.ARRAY_ARRAY_STRING[6][0];
    ARRAY_ARRAY_STRUCTURE_AUTO.ARRAY_ARRAY_STRING[7][1] := ARRAY_ARRAY_STRUCTURE_AUTO.ARRAY_ARRAY_STRING[6][1];
    ARRAY_ARRAY_STRUCTURE_AUTO.ARRAY_ARRAY_STRING[7][2] := ARRAY_ARRAY_STRUCTURE_AUTO.ARRAY_ARRAY_STRING[6][2];
    ARRAY_ARRAY_STRUCTURE_AUTO.ARRAY_ARRAY_STRING[7][3] := ARRAY_ARRAY_STRUCTURE_AUTO.ARRAY_ARRAY_STRING[6][3];
    ARRAY_ARRAY_STRUCTURE_AUTO.ARRAY_ARRAY_STRING[7][4] := ARRAY_ARRAY_STRUCTURE_AUTO.ARRAY_ARRAY_STRING[6][4];
    ARRAY_ARRAY_STRUCTURE_AUTO.ARRAY_ARRAY_STRING[7][5] := ARRAY_ARRAY_STRUCTURE_AUTO.ARRAY_ARRAY_STRING[6][5];
    ARRAY_ARRAY_STRUCTURE_AUTO.ARRAY_ARRAY_STRING[7][6] := ARRAY_ARRAY_STRUCTURE_AUTO.ARRAY_ARRAY_STRING[6][6];
    ARRAY_ARRAY_STRUCTURE_AUTO.ARRAY_ARRAY_STRING[7][7] := ARRAY_ARRAY_STRUCTURE_AUTO.ARRAY_ARRAY_STRING[6][7];
    ARRAY_ARRAY_STRUCTURE_AUTO.ARRAY_ARRAY_STRING[7][8] := ARRAY_ARRAY_STRUCTURE_AUTO.ARRAY_ARRAY_STRING[6][8];
    ARRAY_ARRAY_STRUCTURE_AUTO.ARRAY_ARRAY_STRING[7][9] := ARRAY_ARRAY_STRUCTURE_AUTO.ARRAY_ARRAY_STRING[6][9];

    ARRAY_ARRAY_STRUCTURE_AUTO.ARRAY_ARRAY_TIME[0][0] := ARRAY_ARRAY_STRUCTURE_AUTO.ARRAY_ARRAY_TIME[0][0] + PULSE_TIME;
    ARRAY_ARRAY_STRUCTURE_AUTO.ARRAY_ARRAY_TIME[0][1] := ARRAY_ARRAY_STRUCTURE_AUTO.ARRAY_ARRAY_TIME[0][1] + PULSE_TIME;
    ARRAY_ARRAY_STRUCTURE_AUTO.ARRAY_ARRAY_TIME[0][2] := ARRAY_ARRAY_STRUCTURE_AUTO.ARRAY_ARRAY_TIME[0][2] + PULSE_TIME;
    ARRAY_ARRAY_STRUCTURE_AUTO.ARRAY_ARRAY_TIME[0][3] := ARRAY_ARRAY_STRUCTURE_AUTO.ARRAY_ARRAY_TIME[0][3] + PULSE_TIME;
    ARRAY_ARRAY_STRUCTURE_AUTO.ARRAY_ARRAY_TIME[0][4] := ARRAY_ARRAY_STRUCTURE_AUTO.ARRAY_ARRAY_TIME[0][4] + PULSE_TIME;
    ARRAY_ARRAY_STRUCTURE_AUTO.ARRAY_ARRAY_TIME[0][5] := ARRAY_ARRAY_STRUCTURE_AUTO.ARRAY_ARRAY_TIME[0][5] + PULSE_TIME;
    ARRAY_ARRAY_STRUCTURE_AUTO.ARRAY_ARRAY_TIME[0][6] := ARRAY_ARRAY_STRUCTURE_AUTO.ARRAY_ARRAY_TIME[0][6] + PULSE_TIME;
    ARRAY_ARRAY_STRUCTURE_AUTO.ARRAY_ARRAY_TIME[0][7] := ARRAY_ARRAY_STRUCTURE_AUTO.ARRAY_ARRAY_TIME[0][7] + PULSE_TIME;
    ARRAY_ARRAY_STRUCTURE_AUTO.ARRAY_ARRAY_TIME[0][8] := ARRAY_ARRAY_STRUCTURE_AUTO.ARRAY_ARRAY_TIME[0][6];
    ARRAY_ARRAY_STRUCTURE_AUTO.ARRAY_ARRAY_TIME[0][9] := ARRAY_ARRAY_STRUCTURE_AUTO.ARRAY_ARRAY_TIME[0][7];

    ARRAY_ARRAY_STRUCTURE_AUTO.ARRAY_ARRAY_TIME[1][0] := ARRAY_ARRAY_STRUCTURE_AUTO.ARRAY_ARRAY_TIME[1][0] + PULSE_TIME;
    ARRAY_ARRAY_STRUCTURE_AUTO.ARRAY_ARRAY_TIME[1][1] := ARRAY_ARRAY_STRUCTURE_AUTO.ARRAY_ARRAY_TIME[1][1] + PULSE_TIME;
    ARRAY_ARRAY_STRUCTURE_AUTO.ARRAY_ARRAY_TIME[1][2] := ARRAY_ARRAY_STRUCTURE_AUTO.ARRAY_ARRAY_TIME[1][2] + PULSE_TIME;
    ARRAY_ARRAY_STRUCTURE_AUTO.ARRAY_ARRAY_TIME[1][3] := ARRAY_ARRAY_STRUCTURE_AUTO.ARRAY_ARRAY_TIME[1][3] + PULSE_TIME;
    ARRAY_ARRAY_STRUCTURE_AUTO.ARRAY_ARRAY_TIME[1][4] := ARRAY_ARRAY_STRUCTURE_AUTO.ARRAY_ARRAY_TIME[1][4] + PULSE_TIME;
    ARRAY_ARRAY_STRUCTURE_AUTO.ARRAY_ARRAY_TIME[1][5] := ARRAY_ARRAY_STRUCTURE_AUTO.ARRAY_ARRAY_TIME[1][5] + PULSE_TIME;
    ARRAY_ARRAY_STRUCTURE_AUTO.ARRAY_ARRAY_TIME[1][6] := ARRAY_ARRAY_STRUCTURE_AUTO.ARRAY_ARRAY_TIME[1][6] + PULSE_TIME;
    ARRAY_ARRAY_STRUCTURE_AUTO.ARRAY_ARRAY_TIME[1][7] := ARRAY_ARRAY_STRUCTURE_AUTO.ARRAY_ARRAY_TIME[1][7] + PULSE_TIME;
    ARRAY_ARRAY_STRUCTURE_AUTO.ARRAY_ARRAY_TIME[1][8] := ARRAY_ARRAY_STRUCTURE_AUTO.ARRAY_ARRAY_TIME[1][6];
    ARRAY_ARRAY_STRUCTURE_AUTO.ARRAY_ARRAY_TIME[1][9] := ARRAY_ARRAY_STRUCTURE_AUTO.ARRAY_ARRAY_TIME[1][7];

    ARRAY_ARRAY_STRUCTURE_AUTO.ARRAY_ARRAY_TIME[2][0] := ARRAY_ARRAY_STRUCTURE_AUTO.ARRAY_ARRAY_TIME[2][0] + PULSE_TIME;
    ARRAY_ARRAY_STRUCTURE_AUTO.ARRAY_ARRAY_TIME[2][1] := ARRAY_ARRAY_STRUCTURE_AUTO.ARRAY_ARRAY_TIME[2][1] + PULSE_TIME;
    ARRAY_ARRAY_STRUCTURE_AUTO.ARRAY_ARRAY_TIME[2][2] := ARRAY_ARRAY_STRUCTURE_AUTO.ARRAY_ARRAY_TIME[2][2] + PULSE_TIME;
    ARRAY_ARRAY_STRUCTURE_AUTO.ARRAY_ARRAY_TIME[2][3] := ARRAY_ARRAY_STRUCTURE_AUTO.ARRAY_ARRAY_TIME[2][3] + PULSE_TIME;
    ARRAY_ARRAY_STRUCTURE_AUTO.ARRAY_ARRAY_TIME[2][4] := ARRAY_ARRAY_STRUCTURE_AUTO.ARRAY_ARRAY_TIME[2][4] + PULSE_TIME;
    ARRAY_ARRAY_STRUCTURE_AUTO.ARRAY_ARRAY_TIME[2][5] := ARRAY_ARRAY_STRUCTURE_AUTO.ARRAY_ARRAY_TIME[2][5] + PULSE_TIME;
    ARRAY_ARRAY_STRUCTURE_AUTO.ARRAY_ARRAY_TIME[2][6] := ARRAY_ARRAY_STRUCTURE_AUTO.ARRAY_ARRAY_TIME[2][6] + PULSE_TIME;
    ARRAY_ARRAY_STRUCTURE_AUTO.ARRAY_ARRAY_TIME[2][7] := ARRAY_ARRAY_STRUCTURE_AUTO.ARRAY_ARRAY_TIME[2][7] + PULSE_TIME;
    ARRAY_ARRAY_STRUCTURE_AUTO.ARRAY_ARRAY_TIME[2][8] := ARRAY_ARRAY_STRUCTURE_AUTO.ARRAY_ARRAY_TIME[2][8] + PULSE_TIME;
    ARRAY_ARRAY_STRUCTURE_AUTO.ARRAY_ARRAY_TIME[2][9] := ARRAY_ARRAY_STRUCTURE_AUTO.ARRAY_ARRAY_TIME[2][9] + PULSE_TIME;

    ARRAY_ARRAY_STRUCTURE_AUTO.ARRAY_ARRAY_TIME[3][0] := ARRAY_ARRAY_STRUCTURE_AUTO.ARRAY_ARRAY_TIME[3][0] + PULSE_TIME;
    ARRAY_ARRAY_STRUCTURE_AUTO.ARRAY_ARRAY_TIME[3][1] := ARRAY_ARRAY_STRUCTURE_AUTO.ARRAY_ARRAY_TIME[3][1] + PULSE_TIME;
    ARRAY_ARRAY_STRUCTURE_AUTO.ARRAY_ARRAY_TIME[3][2] := ARRAY_ARRAY_STRUCTURE_AUTO.ARRAY_ARRAY_TIME[3][2] + PULSE_TIME;
    ARRAY_ARRAY_STRUCTURE_AUTO.ARRAY_ARRAY_TIME[3][3] := ARRAY_ARRAY_STRUCTURE_AUTO.ARRAY_ARRAY_TIME[3][3] + PULSE_TIME;
    ARRAY_ARRAY_STRUCTURE_AUTO.ARRAY_ARRAY_TIME[3][4] := ARRAY_ARRAY_STRUCTURE_AUTO.ARRAY_ARRAY_TIME[3][4] + PULSE_TIME;
    ARRAY_ARRAY_STRUCTURE_AUTO.ARRAY_ARRAY_TIME[3][5] := ARRAY_ARRAY_STRUCTURE_AUTO.ARRAY_ARRAY_TIME[3][5] + PULSE_TIME;
    ARRAY_ARRAY_STRUCTURE_AUTO.ARRAY_ARRAY_TIME[3][6] := ARRAY_ARRAY_STRUCTURE_AUTO.ARRAY_ARRAY_TIME[3][6] + PULSE_TIME;
    ARRAY_ARRAY_STRUCTURE_AUTO.ARRAY_ARRAY_TIME[3][7] := ARRAY_ARRAY_STRUCTURE_AUTO.ARRAY_ARRAY_TIME[3][7] + PULSE_TIME;
    ARRAY_ARRAY_STRUCTURE_AUTO.ARRAY_ARRAY_TIME[3][8] := ARRAY_ARRAY_STRUCTURE_AUTO.ARRAY_ARRAY_TIME[3][8] + PULSE_TIME;
    ARRAY_ARRAY_STRUCTURE_AUTO.ARRAY_ARRAY_TIME[3][9] := ARRAY_ARRAY_STRUCTURE_AUTO.ARRAY_ARRAY_TIME[3][9] + PULSE_TIME;

    ARRAY_ARRAY_STRUCTURE_AUTO.ARRAY_ARRAY_TIME[4][0] := ARRAY_ARRAY_STRUCTURE_AUTO.ARRAY_ARRAY_TIME[4][0] + PULSE_TIME;
    ARRAY_ARRAY_STRUCTURE_AUTO.ARRAY_ARRAY_TIME[4][1] := ARRAY_ARRAY_STRUCTURE_AUTO.ARRAY_ARRAY_TIME[4][1] + PULSE_TIME;
    ARRAY_ARRAY_STRUCTURE_AUTO.ARRAY_ARRAY_TIME[4][2] := ARRAY_ARRAY_STRUCTURE_AUTO.ARRAY_ARRAY_TIME[4][2] + PULSE_TIME;
    ARRAY_ARRAY_STRUCTURE_AUTO.ARRAY_ARRAY_TIME[4][3] := ARRAY_ARRAY_STRUCTURE_AUTO.ARRAY_ARRAY_TIME[4][3] + PULSE_TIME;
    ARRAY_ARRAY_STRUCTURE_AUTO.ARRAY_ARRAY_TIME[4][4] := ARRAY_ARRAY_STRUCTURE_AUTO.ARRAY_ARRAY_TIME[4][4] + PULSE_TIME;
    ARRAY_ARRAY_STRUCTURE_AUTO.ARRAY_ARRAY_TIME[4][5] := ARRAY_ARRAY_STRUCTURE_AUTO.ARRAY_ARRAY_TIME[4][5] + PULSE_TIME;
    ARRAY_ARRAY_STRUCTURE_AUTO.ARRAY_ARRAY_TIME[4][6] := ARRAY_ARRAY_STRUCTURE_AUTO.ARRAY_ARRAY_TIME[4][6] + PULSE_TIME;
    ARRAY_ARRAY_STRUCTURE_AUTO.ARRAY_ARRAY_TIME[4][7] := ARRAY_ARRAY_STRUCTURE_AUTO.ARRAY_ARRAY_TIME[4][7] + PULSE_TIME;
    ARRAY_ARRAY_STRUCTURE_AUTO.ARRAY_ARRAY_TIME[4][8] := ARRAY_ARRAY_STRUCTURE_AUTO.ARRAY_ARRAY_TIME[4][8] + PULSE_TIME;
    ARRAY_ARRAY_STRUCTURE_AUTO.ARRAY_ARRAY_TIME[4][9] := ARRAY_ARRAY_STRUCTURE_AUTO.ARRAY_ARRAY_TIME[4][9] + PULSE_TIME;

    ARRAY_ARRAY_STRUCTURE_AUTO.ARRAY_ARRAY_TIME[5][0] := ARRAY_ARRAY_STRUCTURE_AUTO.ARRAY_ARRAY_TIME[5][0] + PULSE_TIME;
    ARRAY_ARRAY_STRUCTURE_AUTO.ARRAY_ARRAY_TIME[5][1] := ARRAY_ARRAY_STRUCTURE_AUTO.ARRAY_ARRAY_TIME[5][1] + PULSE_TIME;
    ARRAY_ARRAY_STRUCTURE_AUTO.ARRAY_ARRAY_TIME[5][2] := ARRAY_ARRAY_STRUCTURE_AUTO.ARRAY_ARRAY_TIME[5][2] + PULSE_TIME;
    ARRAY_ARRAY_STRUCTURE_AUTO.ARRAY_ARRAY_TIME[5][3] := ARRAY_ARRAY_STRUCTURE_AUTO.ARRAY_ARRAY_TIME[5][3] + PULSE_TIME;
    ARRAY_ARRAY_STRUCTURE_AUTO.ARRAY_ARRAY_TIME[5][4] := ARRAY_ARRAY_STRUCTURE_AUTO.ARRAY_ARRAY_TIME[5][4] + PULSE_TIME;
    ARRAY_ARRAY_STRUCTURE_AUTO.ARRAY_ARRAY_TIME[5][5] := ARRAY_ARRAY_STRUCTURE_AUTO.ARRAY_ARRAY_TIME[5][5] + PULSE_TIME;
    ARRAY_ARRAY_STRUCTURE_AUTO.ARRAY_ARRAY_TIME[5][6] := ARRAY_ARRAY_STRUCTURE_AUTO.ARRAY_ARRAY_TIME[5][6] + PULSE_TIME;
    ARRAY_ARRAY_STRUCTURE_AUTO.ARRAY_ARRAY_TIME[5][7] := ARRAY_ARRAY_STRUCTURE_AUTO.ARRAY_ARRAY_TIME[5][7] + PULSE_TIME;
    ARRAY_ARRAY_STRUCTURE_AUTO.ARRAY_ARRAY_TIME[5][8] := ARRAY_ARRAY_STRUCTURE_AUTO.ARRAY_ARRAY_TIME[5][8] + PULSE_TIME;
    ARRAY_ARRAY_STRUCTURE_AUTO.ARRAY_ARRAY_TIME[5][9] := ARRAY_ARRAY_STRUCTURE_AUTO.ARRAY_ARRAY_TIME[5][9] + PULSE_TIME;

    ARRAY_ARRAY_STRUCTURE_AUTO.ARRAY_ARRAY_TIME[6][0] := ARRAY_ARRAY_STRUCTURE_AUTO.ARRAY_ARRAY_TIME[6][0] + PULSE_TIME;
    ARRAY_ARRAY_STRUCTURE_AUTO.ARRAY_ARRAY_TIME[6][1] := ARRAY_ARRAY_STRUCTURE_AUTO.ARRAY_ARRAY_TIME[6][1] + PULSE_TIME;
    ARRAY_ARRAY_STRUCTURE_AUTO.ARRAY_ARRAY_TIME[6][2] := ARRAY_ARRAY_STRUCTURE_AUTO.ARRAY_ARRAY_TIME[6][2] + PULSE_TIME;
    ARRAY_ARRAY_STRUCTURE_AUTO.ARRAY_ARRAY_TIME[6][3] := ARRAY_ARRAY_STRUCTURE_AUTO.ARRAY_ARRAY_TIME[6][3] + PULSE_TIME;
    ARRAY_ARRAY_STRUCTURE_AUTO.ARRAY_ARRAY_TIME[6][4] := ARRAY_ARRAY_STRUCTURE_AUTO.ARRAY_ARRAY_TIME[6][4] + PULSE_TIME;
    ARRAY_ARRAY_STRUCTURE_AUTO.ARRAY_ARRAY_TIME[6][5] := ARRAY_ARRAY_STRUCTURE_AUTO.ARRAY_ARRAY_TIME[6][5] + PULSE_TIME;
    ARRAY_ARRAY_STRUCTURE_AUTO.ARRAY_ARRAY_TIME[6][6] := ARRAY_ARRAY_STRUCTURE_AUTO.ARRAY_ARRAY_TIME[6][6] + PULSE_TIME;
    ARRAY_ARRAY_STRUCTURE_AUTO.ARRAY_ARRAY_TIME[6][7] := ARRAY_ARRAY_STRUCTURE_AUTO.ARRAY_ARRAY_TIME[6][7] + PULSE_TIME;
    ARRAY_ARRAY_STRUCTURE_AUTO.ARRAY_ARRAY_TIME[6][8] := ARRAY_ARRAY_STRUCTURE_AUTO.ARRAY_ARRAY_TIME[6][8] + PULSE_TIME;
    ARRAY_ARRAY_STRUCTURE_AUTO.ARRAY_ARRAY_TIME[6][9] := ARRAY_ARRAY_STRUCTURE_AUTO.ARRAY_ARRAY_TIME[6][9] + PULSE_TIME;

    ARRAY_ARRAY_STRUCTURE_AUTO.ARRAY_ARRAY_TIME[7][0] := ARRAY_ARRAY_STRUCTURE_AUTO.ARRAY_ARRAY_TIME[6][0];
    ARRAY_ARRAY_STRUCTURE_AUTO.ARRAY_ARRAY_TIME[7][1] := ARRAY_ARRAY_STRUCTURE_AUTO.ARRAY_ARRAY_TIME[6][1];
    ARRAY_ARRAY_STRUCTURE_AUTO.ARRAY_ARRAY_TIME[7][2] := ARRAY_ARRAY_STRUCTURE_AUTO.ARRAY_ARRAY_TIME[6][2];
    ARRAY_ARRAY_STRUCTURE_AUTO.ARRAY_ARRAY_TIME[7][3] := ARRAY_ARRAY_STRUCTURE_AUTO.ARRAY_ARRAY_TIME[6][3];
    ARRAY_ARRAY_STRUCTURE_AUTO.ARRAY_ARRAY_TIME[7][4] := ARRAY_ARRAY_STRUCTURE_AUTO.ARRAY_ARRAY_TIME[6][4];
    ARRAY_ARRAY_STRUCTURE_AUTO.ARRAY_ARRAY_TIME[7][5] := ARRAY_ARRAY_STRUCTURE_AUTO.ARRAY_ARRAY_TIME[6][5];
    ARRAY_ARRAY_STRUCTURE_AUTO.ARRAY_ARRAY_TIME[7][6] := ARRAY_ARRAY_STRUCTURE_AUTO.ARRAY_ARRAY_TIME[6][6];
    ARRAY_ARRAY_STRUCTURE_AUTO.ARRAY_ARRAY_TIME[7][7] := ARRAY_ARRAY_STRUCTURE_AUTO.ARRAY_ARRAY_TIME[6][7];
    ARRAY_ARRAY_STRUCTURE_AUTO.ARRAY_ARRAY_TIME[7][8] := ARRAY_ARRAY_STRUCTURE_AUTO.ARRAY_ARRAY_TIME[6][6];
    ARRAY_ARRAY_STRUCTURE_AUTO.ARRAY_ARRAY_TIME[7][9] := ARRAY_ARRAY_STRUCTURE_AUTO.ARRAY_ARRAY_TIME[6][7];

    ARRAY_ARRAY_STRUCTURE_AUTO.ARRAY_ARRAY_UDINT[0][0] := ARRAY_ARRAY_STRUCTURE_AUTO.ARRAY_ARRAY_UDINT[0][0] + 1;
    ARRAY_ARRAY_STRUCTURE_AUTO.ARRAY_ARRAY_UDINT[0][1] := ARRAY_ARRAY_STRUCTURE_AUTO.ARRAY_ARRAY_UDINT[0][1] + 1;
    ARRAY_ARRAY_STRUCTURE_AUTO.ARRAY_ARRAY_UDINT[0][2] := ARRAY_ARRAY_STRUCTURE_AUTO.ARRAY_ARRAY_UDINT[0][2] + 1;
    ARRAY_ARRAY_STRUCTURE_AUTO.ARRAY_ARRAY_UDINT[0][3] := ARRAY_ARRAY_STRUCTURE_AUTO.ARRAY_ARRAY_UDINT[0][3] + 1;
    ARRAY_ARRAY_STRUCTURE_AUTO.ARRAY_ARRAY_UDINT[0][4] := ARRAY_ARRAY_STRUCTURE_AUTO.ARRAY_ARRAY_UDINT[0][4] + 1;
    ARRAY_ARRAY_STRUCTURE_AUTO.ARRAY_ARRAY_UDINT[0][5] := ARRAY_ARRAY_STRUCTURE_AUTO.ARRAY_ARRAY_UDINT[0][5] + 1;
    ARRAY_ARRAY_STRUCTURE_AUTO.ARRAY_ARRAY_UDINT[0][6] := ARRAY_ARRAY_STRUCTURE_AUTO.ARRAY_ARRAY_UDINT[0][6] + 1;
    ARRAY_ARRAY_STRUCTURE_AUTO.ARRAY_ARRAY_UDINT[0][7] := ARRAY_ARRAY_STRUCTURE_AUTO.ARRAY_ARRAY_UDINT[0][7] + 1;
    ARRAY_ARRAY_STRUCTURE_AUTO.ARRAY_ARRAY_UDINT[0][8] := ARRAY_ARRAY_STRUCTURE_AUTO.ARRAY_ARRAY_UDINT[0][6];
    ARRAY_ARRAY_STRUCTURE_AUTO.ARRAY_ARRAY_UDINT[0][9] := ARRAY_ARRAY_STRUCTURE_AUTO.ARRAY_ARRAY_UDINT[0][7];

    ARRAY_ARRAY_STRUCTURE_AUTO.ARRAY_ARRAY_UDINT[1][0] := ARRAY_ARRAY_STRUCTURE_AUTO.ARRAY_ARRAY_UDINT[1][0] + 1;
    ARRAY_ARRAY_STRUCTURE_AUTO.ARRAY_ARRAY_UDINT[1][1] := ARRAY_ARRAY_STRUCTURE_AUTO.ARRAY_ARRAY_UDINT[1][1] + 1;
    ARRAY_ARRAY_STRUCTURE_AUTO.ARRAY_ARRAY_UDINT[1][2] := ARRAY_ARRAY_STRUCTURE_AUTO.ARRAY_ARRAY_UDINT[1][2] + 1;
    ARRAY_ARRAY_STRUCTURE_AUTO.ARRAY_ARRAY_UDINT[1][3] := ARRAY_ARRAY_STRUCTURE_AUTO.ARRAY_ARRAY_UDINT[1][3] + 1;
    ARRAY_ARRAY_STRUCTURE_AUTO.ARRAY_ARRAY_UDINT[1][4] := ARRAY_ARRAY_STRUCTURE_AUTO.ARRAY_ARRAY_UDINT[1][4] + 1;
    ARRAY_ARRAY_STRUCTURE_AUTO.ARRAY_ARRAY_UDINT[1][5] := ARRAY_ARRAY_STRUCTURE_AUTO.ARRAY_ARRAY_UDINT[1][5] + 1;
    ARRAY_ARRAY_STRUCTURE_AUTO.ARRAY_ARRAY_UDINT[1][6] := ARRAY_ARRAY_STRUCTURE_AUTO.ARRAY_ARRAY_UDINT[1][6] + 1;
    ARRAY_ARRAY_STRUCTURE_AUTO.ARRAY_ARRAY_UDINT[1][7] := ARRAY_ARRAY_STRUCTURE_AUTO.ARRAY_ARRAY_UDINT[1][7] + 1;
    ARRAY_ARRAY_STRUCTURE_AUTO.ARRAY_ARRAY_UDINT[1][8] := ARRAY_ARRAY_STRUCTURE_AUTO.ARRAY_ARRAY_UDINT[1][6];
    ARRAY_ARRAY_STRUCTURE_AUTO.ARRAY_ARRAY_UDINT[1][9] := ARRAY_ARRAY_STRUCTURE_AUTO.ARRAY_ARRAY_UDINT[1][7];

    ARRAY_ARRAY_STRUCTURE_AUTO.ARRAY_ARRAY_UDINT[2][0] := ARRAY_ARRAY_STRUCTURE_AUTO.ARRAY_ARRAY_UDINT[2][0] + 1;
    ARRAY_ARRAY_STRUCTURE_AUTO.ARRAY_ARRAY_UDINT[2][1] := ARRAY_ARRAY_STRUCTURE_AUTO.ARRAY_ARRAY_UDINT[2][1] + 1;
    ARRAY_ARRAY_STRUCTURE_AUTO.ARRAY_ARRAY_UDINT[2][2] := ARRAY_ARRAY_STRUCTURE_AUTO.ARRAY_ARRAY_UDINT[2][2] + 1;
    ARRAY_ARRAY_STRUCTURE_AUTO.ARRAY_ARRAY_UDINT[2][3] := ARRAY_ARRAY_STRUCTURE_AUTO.ARRAY_ARRAY_UDINT[2][3] + 1;
    ARRAY_ARRAY_STRUCTURE_AUTO.ARRAY_ARRAY_UDINT[2][4] := ARRAY_ARRAY_STRUCTURE_AUTO.ARRAY_ARRAY_UDINT[2][4] + 1;
    ARRAY_ARRAY_STRUCTURE_AUTO.ARRAY_ARRAY_UDINT[2][5] := ARRAY_ARRAY_STRUCTURE_AUTO.ARRAY_ARRAY_UDINT[2][5] + 1;
    ARRAY_ARRAY_STRUCTURE_AUTO.ARRAY_ARRAY_UDINT[2][6] := ARRAY_ARRAY_STRUCTURE_AUTO.ARRAY_ARRAY_UDINT[2][6] + 1;
    ARRAY_ARRAY_STRUCTURE_AUTO.ARRAY_ARRAY_UDINT[2][7] := ARRAY_ARRAY_STRUCTURE_AUTO.ARRAY_ARRAY_UDINT[2][7] + 1;
    ARRAY_ARRAY_STRUCTURE_AUTO.ARRAY_ARRAY_UDINT[2][8] := ARRAY_ARRAY_STRUCTURE_AUTO.ARRAY_ARRAY_UDINT[2][8] + 1;
    ARRAY_ARRAY_STRUCTURE_AUTO.ARRAY_ARRAY_UDINT[2][9] := ARRAY_ARRAY_STRUCTURE_AUTO.ARRAY_ARRAY_UDINT[2][9] + 1;

    ARRAY_ARRAY_STRUCTURE_AUTO.ARRAY_ARRAY_UDINT[3][0] := ARRAY_ARRAY_STRUCTURE_AUTO.ARRAY_ARRAY_UDINT[3][0] + 1;
    ARRAY_ARRAY_STRUCTURE_AUTO.ARRAY_ARRAY_UDINT[3][1] := ARRAY_ARRAY_STRUCTURE_AUTO.ARRAY_ARRAY_UDINT[3][1] + 1;
    ARRAY_ARRAY_STRUCTURE_AUTO.ARRAY_ARRAY_UDINT[3][2] := ARRAY_ARRAY_STRUCTURE_AUTO.ARRAY_ARRAY_UDINT[3][2] + 1;
    ARRAY_ARRAY_STRUCTURE_AUTO.ARRAY_ARRAY_UDINT[3][3] := ARRAY_ARRAY_STRUCTURE_AUTO.ARRAY_ARRAY_UDINT[3][3] + 1;
    ARRAY_ARRAY_STRUCTURE_AUTO.ARRAY_ARRAY_UDINT[3][4] := ARRAY_ARRAY_STRUCTURE_AUTO.ARRAY_ARRAY_UDINT[3][4] + 1;
    ARRAY_ARRAY_STRUCTURE_AUTO.ARRAY_ARRAY_UDINT[3][5] := ARRAY_ARRAY_STRUCTURE_AUTO.ARRAY_ARRAY_UDINT[3][5] + 1;
    ARRAY_ARRAY_STRUCTURE_AUTO.ARRAY_ARRAY_UDINT[3][6] := ARRAY_ARRAY_STRUCTURE_AUTO.ARRAY_ARRAY_UDINT[3][6] + 1;
    ARRAY_ARRAY_STRUCTURE_AUTO.ARRAY_ARRAY_UDINT[3][7] := ARRAY_ARRAY_STRUCTURE_AUTO.ARRAY_ARRAY_UDINT[3][7] + 1;
    ARRAY_ARRAY_STRUCTURE_AUTO.ARRAY_ARRAY_UDINT[3][8] := ARRAY_ARRAY_STRUCTURE_AUTO.ARRAY_ARRAY_UDINT[3][8] + 1;
    ARRAY_ARRAY_STRUCTURE_AUTO.ARRAY_ARRAY_UDINT[3][9] := ARRAY_ARRAY_STRUCTURE_AUTO.ARRAY_ARRAY_UDINT[3][9] + 1;

    ARRAY_ARRAY_STRUCTURE_AUTO.ARRAY_ARRAY_UDINT[4][0] := ARRAY_ARRAY_STRUCTURE_AUTO.ARRAY_ARRAY_UDINT[4][0] + 1;
    ARRAY_ARRAY_STRUCTURE_AUTO.ARRAY_ARRAY_UDINT[4][1] := ARRAY_ARRAY_STRUCTURE_AUTO.ARRAY_ARRAY_UDINT[4][1] + 1;
    ARRAY_ARRAY_STRUCTURE_AUTO.ARRAY_ARRAY_UDINT[4][2] := ARRAY_ARRAY_STRUCTURE_AUTO.ARRAY_ARRAY_UDINT[4][2] + 1;
    ARRAY_ARRAY_STRUCTURE_AUTO.ARRAY_ARRAY_UDINT[4][3] := ARRAY_ARRAY_STRUCTURE_AUTO.ARRAY_ARRAY_UDINT[4][3] + 1;
    ARRAY_ARRAY_STRUCTURE_AUTO.ARRAY_ARRAY_UDINT[4][4] := ARRAY_ARRAY_STRUCTURE_AUTO.ARRAY_ARRAY_UDINT[4][4] + 1;
    ARRAY_ARRAY_STRUCTURE_AUTO.ARRAY_ARRAY_UDINT[4][5] := ARRAY_ARRAY_STRUCTURE_AUTO.ARRAY_ARRAY_UDINT[4][5] + 1;
    ARRAY_ARRAY_STRUCTURE_AUTO.ARRAY_ARRAY_UDINT[4][6] := ARRAY_ARRAY_STRUCTURE_AUTO.ARRAY_ARRAY_UDINT[4][6] + 1;
    ARRAY_ARRAY_STRUCTURE_AUTO.ARRAY_ARRAY_UDINT[4][7] := ARRAY_ARRAY_STRUCTURE_AUTO.ARRAY_ARRAY_UDINT[4][7] + 1;
    ARRAY_ARRAY_STRUCTURE_AUTO.ARRAY_ARRAY_UDINT[4][8] := ARRAY_ARRAY_STRUCTURE_AUTO.ARRAY_ARRAY_UDINT[4][8] + 1;
    ARRAY_ARRAY_STRUCTURE_AUTO.ARRAY_ARRAY_UDINT[4][9] := ARRAY_ARRAY_STRUCTURE_AUTO.ARRAY_ARRAY_UDINT[4][9] + 1;

    ARRAY_ARRAY_STRUCTURE_AUTO.ARRAY_ARRAY_UDINT[5][0] := ARRAY_ARRAY_STRUCTURE_AUTO.ARRAY_ARRAY_UDINT[5][0] + 1;
    ARRAY_ARRAY_STRUCTURE_AUTO.ARRAY_ARRAY_UDINT[5][1] := ARRAY_ARRAY_STRUCTURE_AUTO.ARRAY_ARRAY_UDINT[5][1] + 1;
    ARRAY_ARRAY_STRUCTURE_AUTO.ARRAY_ARRAY_UDINT[5][2] := ARRAY_ARRAY_STRUCTURE_AUTO.ARRAY_ARRAY_UDINT[5][2] + 1;
    ARRAY_ARRAY_STRUCTURE_AUTO.ARRAY_ARRAY_UDINT[5][3] := ARRAY_ARRAY_STRUCTURE_AUTO.ARRAY_ARRAY_UDINT[5][3] + 1;
    ARRAY_ARRAY_STRUCTURE_AUTO.ARRAY_ARRAY_UDINT[5][4] := ARRAY_ARRAY_STRUCTURE_AUTO.ARRAY_ARRAY_UDINT[5][4] + 1;
    ARRAY_ARRAY_STRUCTURE_AUTO.ARRAY_ARRAY_UDINT[5][5] := ARRAY_ARRAY_STRUCTURE_AUTO.ARRAY_ARRAY_UDINT[5][5] + 1;
    ARRAY_ARRAY_STRUCTURE_AUTO.ARRAY_ARRAY_UDINT[5][6] := ARRAY_ARRAY_STRUCTURE_AUTO.ARRAY_ARRAY_UDINT[5][6] + 1;
    ARRAY_ARRAY_STRUCTURE_AUTO.ARRAY_ARRAY_UDINT[5][7] := ARRAY_ARRAY_STRUCTURE_AUTO.ARRAY_ARRAY_UDINT[5][7] + 1;
    ARRAY_ARRAY_STRUCTURE_AUTO.ARRAY_ARRAY_UDINT[5][8] := ARRAY_ARRAY_STRUCTURE_AUTO.ARRAY_ARRAY_UDINT[5][8] + 1;
    ARRAY_ARRAY_STRUCTURE_AUTO.ARRAY_ARRAY_UDINT[5][9] := ARRAY_ARRAY_STRUCTURE_AUTO.ARRAY_ARRAY_UDINT[5][9] + 1;

    ARRAY_ARRAY_STRUCTURE_AUTO.ARRAY_ARRAY_UDINT[6][0] := ARRAY_ARRAY_STRUCTURE_AUTO.ARRAY_ARRAY_UDINT[6][0] + 1;
    ARRAY_ARRAY_STRUCTURE_AUTO.ARRAY_ARRAY_UDINT[6][1] := ARRAY_ARRAY_STRUCTURE_AUTO.ARRAY_ARRAY_UDINT[6][1] + 1;
    ARRAY_ARRAY_STRUCTURE_AUTO.ARRAY_ARRAY_UDINT[6][2] := ARRAY_ARRAY_STRUCTURE_AUTO.ARRAY_ARRAY_UDINT[6][2] + 1;
    ARRAY_ARRAY_STRUCTURE_AUTO.ARRAY_ARRAY_UDINT[6][3] := ARRAY_ARRAY_STRUCTURE_AUTO.ARRAY_ARRAY_UDINT[6][3] + 1;
    ARRAY_ARRAY_STRUCTURE_AUTO.ARRAY_ARRAY_UDINT[6][4] := ARRAY_ARRAY_STRUCTURE_AUTO.ARRAY_ARRAY_UDINT[6][4] + 1;
    ARRAY_ARRAY_STRUCTURE_AUTO.ARRAY_ARRAY_UDINT[6][5] := ARRAY_ARRAY_STRUCTURE_AUTO.ARRAY_ARRAY_UDINT[6][5] + 1;
    ARRAY_ARRAY_STRUCTURE_AUTO.ARRAY_ARRAY_UDINT[6][6] := ARRAY_ARRAY_STRUCTURE_AUTO.ARRAY_ARRAY_UDINT[6][6] + 1;
    ARRAY_ARRAY_STRUCTURE_AUTO.ARRAY_ARRAY_UDINT[6][7] := ARRAY_ARRAY_STRUCTURE_AUTO.ARRAY_ARRAY_UDINT[6][7] + 1;
    ARRAY_ARRAY_STRUCTURE_AUTO.ARRAY_ARRAY_UDINT[6][8] := ARRAY_ARRAY_STRUCTURE_AUTO.ARRAY_ARRAY_UDINT[6][8] + 1;
    ARRAY_ARRAY_STRUCTURE_AUTO.ARRAY_ARRAY_UDINT[6][9] := ARRAY_ARRAY_STRUCTURE_AUTO.ARRAY_ARRAY_UDINT[6][9] + 1;

    ARRAY_ARRAY_STRUCTURE_AUTO.ARRAY_ARRAY_UDINT[7][0] := ARRAY_ARRAY_STRUCTURE_AUTO.ARRAY_ARRAY_UDINT[6][0];
    ARRAY_ARRAY_STRUCTURE_AUTO.ARRAY_ARRAY_UDINT[7][1] := ARRAY_ARRAY_STRUCTURE_AUTO.ARRAY_ARRAY_UDINT[6][1];
    ARRAY_ARRAY_STRUCTURE_AUTO.ARRAY_ARRAY_UDINT[7][2] := ARRAY_ARRAY_STRUCTURE_AUTO.ARRAY_ARRAY_UDINT[6][2];
    ARRAY_ARRAY_STRUCTURE_AUTO.ARRAY_ARRAY_UDINT[7][3] := ARRAY_ARRAY_STRUCTURE_AUTO.ARRAY_ARRAY_UDINT[6][3];
    ARRAY_ARRAY_STRUCTURE_AUTO.ARRAY_ARRAY_UDINT[7][4] := ARRAY_ARRAY_STRUCTURE_AUTO.ARRAY_ARRAY_UDINT[6][4];
    ARRAY_ARRAY_STRUCTURE_AUTO.ARRAY_ARRAY_UDINT[7][5] := ARRAY_ARRAY_STRUCTURE_AUTO.ARRAY_ARRAY_UDINT[6][5];
    ARRAY_ARRAY_STRUCTURE_AUTO.ARRAY_ARRAY_UDINT[7][6] := ARRAY_ARRAY_STRUCTURE_AUTO.ARRAY_ARRAY_UDINT[6][6];
    ARRAY_ARRAY_STRUCTURE_AUTO.ARRAY_ARRAY_UDINT[7][7] := ARRAY_ARRAY_STRUCTURE_AUTO.ARRAY_ARRAY_UDINT[6][7];
    ARRAY_ARRAY_STRUCTURE_AUTO.ARRAY_ARRAY_UDINT[7][8] := ARRAY_ARRAY_STRUCTURE_AUTO.ARRAY_ARRAY_UDINT[6][8];
    ARRAY_ARRAY_STRUCTURE_AUTO.ARRAY_ARRAY_UDINT[7][9] := ARRAY_ARRAY_STRUCTURE_AUTO.ARRAY_ARRAY_UDINT[6][9];

    ARRAY_ARRAY_STRUCTURE_AUTO.ARRAY_ARRAY_UINT[0][0] := ARRAY_ARRAY_STRUCTURE_AUTO.ARRAY_ARRAY_UINT[0][0] + 1;
    ARRAY_ARRAY_STRUCTURE_AUTO.ARRAY_ARRAY_UINT[0][1] := ARRAY_ARRAY_STRUCTURE_AUTO.ARRAY_ARRAY_UINT[0][1] + 1;
    ARRAY_ARRAY_STRUCTURE_AUTO.ARRAY_ARRAY_UINT[0][2] := ARRAY_ARRAY_STRUCTURE_AUTO.ARRAY_ARRAY_UINT[0][2] + 1;
    ARRAY_ARRAY_STRUCTURE_AUTO.ARRAY_ARRAY_UINT[0][3] := ARRAY_ARRAY_STRUCTURE_AUTO.ARRAY_ARRAY_UINT[0][3] + 1;
    ARRAY_ARRAY_STRUCTURE_AUTO.ARRAY_ARRAY_UINT[0][4] := ARRAY_ARRAY_STRUCTURE_AUTO.ARRAY_ARRAY_UINT[0][4] + 1;
    ARRAY_ARRAY_STRUCTURE_AUTO.ARRAY_ARRAY_UINT[0][5] := ARRAY_ARRAY_STRUCTURE_AUTO.ARRAY_ARRAY_UINT[0][5] + 1;
    ARRAY_ARRAY_STRUCTURE_AUTO.ARRAY_ARRAY_UINT[0][6] := ARRAY_ARRAY_STRUCTURE_AUTO.ARRAY_ARRAY_UINT[0][6] + 1;
    ARRAY_ARRAY_STRUCTURE_AUTO.ARRAY_ARRAY_UINT[0][7] := ARRAY_ARRAY_STRUCTURE_AUTO.ARRAY_ARRAY_UINT[0][7] + 1;
    ARRAY_ARRAY_STRUCTURE_AUTO.ARRAY_ARRAY_UINT[0][8] := ARRAY_ARRAY_STRUCTURE_AUTO.ARRAY_ARRAY_UINT[0][6];
    ARRAY_ARRAY_STRUCTURE_AUTO.ARRAY_ARRAY_UINT[0][9] := ARRAY_ARRAY_STRUCTURE_AUTO.ARRAY_ARRAY_UINT[0][7];

    ARRAY_ARRAY_STRUCTURE_AUTO.ARRAY_ARRAY_UINT[1][0] := ARRAY_ARRAY_STRUCTURE_AUTO.ARRAY_ARRAY_UINT[1][0] + 1;
    ARRAY_ARRAY_STRUCTURE_AUTO.ARRAY_ARRAY_UINT[1][1] := ARRAY_ARRAY_STRUCTURE_AUTO.ARRAY_ARRAY_UINT[1][1] + 1;
    ARRAY_ARRAY_STRUCTURE_AUTO.ARRAY_ARRAY_UINT[1][2] := ARRAY_ARRAY_STRUCTURE_AUTO.ARRAY_ARRAY_UINT[1][2] + 1;
    ARRAY_ARRAY_STRUCTURE_AUTO.ARRAY_ARRAY_UINT[1][3] := ARRAY_ARRAY_STRUCTURE_AUTO.ARRAY_ARRAY_UINT[1][3] + 1;
    ARRAY_ARRAY_STRUCTURE_AUTO.ARRAY_ARRAY_UINT[1][4] := ARRAY_ARRAY_STRUCTURE_AUTO.ARRAY_ARRAY_UINT[1][4] + 1;
    ARRAY_ARRAY_STRUCTURE_AUTO.ARRAY_ARRAY_UINT[1][5] := ARRAY_ARRAY_STRUCTURE_AUTO.ARRAY_ARRAY_UINT[1][5] + 1;
    ARRAY_ARRAY_STRUCTURE_AUTO.ARRAY_ARRAY_UINT[1][6] := ARRAY_ARRAY_STRUCTURE_AUTO.ARRAY_ARRAY_UINT[1][6] + 1;
    ARRAY_ARRAY_STRUCTURE_AUTO.ARRAY_ARRAY_UINT[1][7] := ARRAY_ARRAY_STRUCTURE_AUTO.ARRAY_ARRAY_UINT[1][7] + 1;
    ARRAY_ARRAY_STRUCTURE_AUTO.ARRAY_ARRAY_UINT[1][8] := ARRAY_ARRAY_STRUCTURE_AUTO.ARRAY_ARRAY_UINT[1][6];
    ARRAY_ARRAY_STRUCTURE_AUTO.ARRAY_ARRAY_UINT[1][9] := ARRAY_ARRAY_STRUCTURE_AUTO.ARRAY_ARRAY_UINT[1][7];

    ARRAY_ARRAY_STRUCTURE_AUTO.ARRAY_ARRAY_UINT[2][0] := ARRAY_ARRAY_STRUCTURE_AUTO.ARRAY_ARRAY_UINT[2][0] + 1;
    ARRAY_ARRAY_STRUCTURE_AUTO.ARRAY_ARRAY_UINT[2][1] := ARRAY_ARRAY_STRUCTURE_AUTO.ARRAY_ARRAY_UINT[2][1] + 1;
    ARRAY_ARRAY_STRUCTURE_AUTO.ARRAY_ARRAY_UINT[2][2] := ARRAY_ARRAY_STRUCTURE_AUTO.ARRAY_ARRAY_UINT[2][2] + 1;
    ARRAY_ARRAY_STRUCTURE_AUTO.ARRAY_ARRAY_UINT[2][3] := ARRAY_ARRAY_STRUCTURE_AUTO.ARRAY_ARRAY_UINT[2][3] + 1;
    ARRAY_ARRAY_STRUCTURE_AUTO.ARRAY_ARRAY_UINT[2][4] := ARRAY_ARRAY_STRUCTURE_AUTO.ARRAY_ARRAY_UINT[2][4] + 1;
    ARRAY_ARRAY_STRUCTURE_AUTO.ARRAY_ARRAY_UINT[2][5] := ARRAY_ARRAY_STRUCTURE_AUTO.ARRAY_ARRAY_UINT[2][5] + 1;
    ARRAY_ARRAY_STRUCTURE_AUTO.ARRAY_ARRAY_UINT[2][6] := ARRAY_ARRAY_STRUCTURE_AUTO.ARRAY_ARRAY_UINT[2][6] + 1;
    ARRAY_ARRAY_STRUCTURE_AUTO.ARRAY_ARRAY_UINT[2][7] := ARRAY_ARRAY_STRUCTURE_AUTO.ARRAY_ARRAY_UINT[2][7] + 1;
    ARRAY_ARRAY_STRUCTURE_AUTO.ARRAY_ARRAY_UINT[2][8] := ARRAY_ARRAY_STRUCTURE_AUTO.ARRAY_ARRAY_UINT[2][8] + 1;
    ARRAY_ARRAY_STRUCTURE_AUTO.ARRAY_ARRAY_UINT[2][9] := ARRAY_ARRAY_STRUCTURE_AUTO.ARRAY_ARRAY_UINT[2][9] + 1;

    ARRAY_ARRAY_STRUCTURE_AUTO.ARRAY_ARRAY_UINT[3][0] := ARRAY_ARRAY_STRUCTURE_AUTO.ARRAY_ARRAY_UINT[3][0] + 1;
    ARRAY_ARRAY_STRUCTURE_AUTO.ARRAY_ARRAY_UINT[3][1] := ARRAY_ARRAY_STRUCTURE_AUTO.ARRAY_ARRAY_UINT[3][1] + 1;
    ARRAY_ARRAY_STRUCTURE_AUTO.ARRAY_ARRAY_UINT[3][2] := ARRAY_ARRAY_STRUCTURE_AUTO.ARRAY_ARRAY_UINT[3][2] + 1;
    ARRAY_ARRAY_STRUCTURE_AUTO.ARRAY_ARRAY_UINT[3][3] := ARRAY_ARRAY_STRUCTURE_AUTO.ARRAY_ARRAY_UINT[3][3] + 1;
    ARRAY_ARRAY_STRUCTURE_AUTO.ARRAY_ARRAY_UINT[3][4] := ARRAY_ARRAY_STRUCTURE_AUTO.ARRAY_ARRAY_UINT[3][4] + 1;
    ARRAY_ARRAY_STRUCTURE_AUTO.ARRAY_ARRAY_UINT[3][5] := ARRAY_ARRAY_STRUCTURE_AUTO.ARRAY_ARRAY_UINT[3][5] + 1;
    ARRAY_ARRAY_STRUCTURE_AUTO.ARRAY_ARRAY_UINT[3][6] := ARRAY_ARRAY_STRUCTURE_AUTO.ARRAY_ARRAY_UINT[3][6] + 1;
    ARRAY_ARRAY_STRUCTURE_AUTO.ARRAY_ARRAY_UINT[3][7] := ARRAY_ARRAY_STRUCTURE_AUTO.ARRAY_ARRAY_UINT[3][7] + 1;
    ARRAY_ARRAY_STRUCTURE_AUTO.ARRAY_ARRAY_UINT[3][8] := ARRAY_ARRAY_STRUCTURE_AUTO.ARRAY_ARRAY_UINT[3][8] + 1;
    ARRAY_ARRAY_STRUCTURE_AUTO.ARRAY_ARRAY_UINT[3][9] := ARRAY_ARRAY_STRUCTURE_AUTO.ARRAY_ARRAY_UINT[3][9] + 1;

    ARRAY_ARRAY_STRUCTURE_AUTO.ARRAY_ARRAY_UINT[4][0] := ARRAY_ARRAY_STRUCTURE_AUTO.ARRAY_ARRAY_UINT[4][0] + 1;
    ARRAY_ARRAY_STRUCTURE_AUTO.ARRAY_ARRAY_UINT[4][1] := ARRAY_ARRAY_STRUCTURE_AUTO.ARRAY_ARRAY_UINT[4][1] + 1;
    ARRAY_ARRAY_STRUCTURE_AUTO.ARRAY_ARRAY_UINT[4][2] := ARRAY_ARRAY_STRUCTURE_AUTO.ARRAY_ARRAY_UINT[4][2] + 1;
    ARRAY_ARRAY_STRUCTURE_AUTO.ARRAY_ARRAY_UINT[4][3] := ARRAY_ARRAY_STRUCTURE_AUTO.ARRAY_ARRAY_UINT[4][3] + 1;
    ARRAY_ARRAY_STRUCTURE_AUTO.ARRAY_ARRAY_UINT[4][4] := ARRAY_ARRAY_STRUCTURE_AUTO.ARRAY_ARRAY_UINT[4][4] + 1;
    ARRAY_ARRAY_STRUCTURE_AUTO.ARRAY_ARRAY_UINT[4][5] := ARRAY_ARRAY_STRUCTURE_AUTO.ARRAY_ARRAY_UINT[4][5] + 1;
    ARRAY_ARRAY_STRUCTURE_AUTO.ARRAY_ARRAY_UINT[4][6] := ARRAY_ARRAY_STRUCTURE_AUTO.ARRAY_ARRAY_UINT[4][6] + 1;
    ARRAY_ARRAY_STRUCTURE_AUTO.ARRAY_ARRAY_UINT[4][7] := ARRAY_ARRAY_STRUCTURE_AUTO.ARRAY_ARRAY_UINT[4][7] + 1;
    ARRAY_ARRAY_STRUCTURE_AUTO.ARRAY_ARRAY_UINT[4][8] := ARRAY_ARRAY_STRUCTURE_AUTO.ARRAY_ARRAY_UINT[4][8] + 1;
    ARRAY_ARRAY_STRUCTURE_AUTO.ARRAY_ARRAY_UINT[4][9] := ARRAY_ARRAY_STRUCTURE_AUTO.ARRAY_ARRAY_UINT[4][9] + 1;

    ARRAY_ARRAY_STRUCTURE_AUTO.ARRAY_ARRAY_UINT[5][0] := ARRAY_ARRAY_STRUCTURE_AUTO.ARRAY_ARRAY_UINT[5][0] + 1;
    ARRAY_ARRAY_STRUCTURE_AUTO.ARRAY_ARRAY_UINT[5][1] := ARRAY_ARRAY_STRUCTURE_AUTO.ARRAY_ARRAY_UINT[5][1] + 1;
    ARRAY_ARRAY_STRUCTURE_AUTO.ARRAY_ARRAY_UINT[5][2] := ARRAY_ARRAY_STRUCTURE_AUTO.ARRAY_ARRAY_UINT[5][2] + 1;
    ARRAY_ARRAY_STRUCTURE_AUTO.ARRAY_ARRAY_UINT[5][3] := ARRAY_ARRAY_STRUCTURE_AUTO.ARRAY_ARRAY_UINT[5][3] + 1;
    ARRAY_ARRAY_STRUCTURE_AUTO.ARRAY_ARRAY_UINT[5][4] := ARRAY_ARRAY_STRUCTURE_AUTO.ARRAY_ARRAY_UINT[5][4] + 1;
    ARRAY_ARRAY_STRUCTURE_AUTO.ARRAY_ARRAY_UINT[5][5] := ARRAY_ARRAY_STRUCTURE_AUTO.ARRAY_ARRAY_UINT[5][5] + 1;
    ARRAY_ARRAY_STRUCTURE_AUTO.ARRAY_ARRAY_UINT[5][6] := ARRAY_ARRAY_STRUCTURE_AUTO.ARRAY_ARRAY_UINT[5][6] + 1;
    ARRAY_ARRAY_STRUCTURE_AUTO.ARRAY_ARRAY_UINT[5][7] := ARRAY_ARRAY_STRUCTURE_AUTO.ARRAY_ARRAY_UINT[5][7] + 1;
    ARRAY_ARRAY_STRUCTURE_AUTO.ARRAY_ARRAY_UINT[5][8] := ARRAY_ARRAY_STRUCTURE_AUTO.ARRAY_ARRAY_UINT[5][8] + 1;
    ARRAY_ARRAY_STRUCTURE_AUTO.ARRAY_ARRAY_UINT[5][9] := ARRAY_ARRAY_STRUCTURE_AUTO.ARRAY_ARRAY_UINT[5][9] + 1;

    ARRAY_ARRAY_STRUCTURE_AUTO.ARRAY_ARRAY_UINT[6][0] := ARRAY_ARRAY_STRUCTURE_AUTO.ARRAY_ARRAY_UINT[6][0] + 1;
    ARRAY_ARRAY_STRUCTURE_AUTO.ARRAY_ARRAY_UINT[6][1] := ARRAY_ARRAY_STRUCTURE_AUTO.ARRAY_ARRAY_UINT[6][1] + 1;
    ARRAY_ARRAY_STRUCTURE_AUTO.ARRAY_ARRAY_UINT[6][2] := ARRAY_ARRAY_STRUCTURE_AUTO.ARRAY_ARRAY_UINT[6][2] + 1;
    ARRAY_ARRAY_STRUCTURE_AUTO.ARRAY_ARRAY_UINT[6][3] := ARRAY_ARRAY_STRUCTURE_AUTO.ARRAY_ARRAY_UINT[6][3] + 1;
    ARRAY_ARRAY_STRUCTURE_AUTO.ARRAY_ARRAY_UINT[6][4] := ARRAY_ARRAY_STRUCTURE_AUTO.ARRAY_ARRAY_UINT[6][4] + 1;
    ARRAY_ARRAY_STRUCTURE_AUTO.ARRAY_ARRAY_UINT[6][5] := ARRAY_ARRAY_STRUCTURE_AUTO.ARRAY_ARRAY_UINT[6][5] + 1;
    ARRAY_ARRAY_STRUCTURE_AUTO.ARRAY_ARRAY_UINT[6][6] := ARRAY_ARRAY_STRUCTURE_AUTO.ARRAY_ARRAY_UINT[6][6] + 1;
    ARRAY_ARRAY_STRUCTURE_AUTO.ARRAY_ARRAY_UINT[6][7] := ARRAY_ARRAY_STRUCTURE_AUTO.ARRAY_ARRAY_UINT[6][7] + 1;
    ARRAY_ARRAY_STRUCTURE_AUTO.ARRAY_ARRAY_UINT[6][8] := ARRAY_ARRAY_STRUCTURE_AUTO.ARRAY_ARRAY_UINT[6][8] + 1;
    ARRAY_ARRAY_STRUCTURE_AUTO.ARRAY_ARRAY_UINT[6][9] := ARRAY_ARRAY_STRUCTURE_AUTO.ARRAY_ARRAY_UINT[6][9] + 1;

    ARRAY_ARRAY_STRUCTURE_AUTO.ARRAY_ARRAY_UINT[7][0] := ARRAY_ARRAY_STRUCTURE_AUTO.ARRAY_ARRAY_UINT[6][0];
    ARRAY_ARRAY_STRUCTURE_AUTO.ARRAY_ARRAY_UINT[7][1] := ARRAY_ARRAY_STRUCTURE_AUTO.ARRAY_ARRAY_UINT[6][1];
    ARRAY_ARRAY_STRUCTURE_AUTO.ARRAY_ARRAY_UINT[7][2] := ARRAY_ARRAY_STRUCTURE_AUTO.ARRAY_ARRAY_UINT[6][2];
    ARRAY_ARRAY_STRUCTURE_AUTO.ARRAY_ARRAY_UINT[7][3] := ARRAY_ARRAY_STRUCTURE_AUTO.ARRAY_ARRAY_UINT[6][3];
    ARRAY_ARRAY_STRUCTURE_AUTO.ARRAY_ARRAY_UINT[7][4] := ARRAY_ARRAY_STRUCTURE_AUTO.ARRAY_ARRAY_UINT[6][4];
    ARRAY_ARRAY_STRUCTURE_AUTO.ARRAY_ARRAY_UINT[7][5] := ARRAY_ARRAY_STRUCTURE_AUTO.ARRAY_ARRAY_UINT[6][5];
    ARRAY_ARRAY_STRUCTURE_AUTO.ARRAY_ARRAY_UINT[7][6] := ARRAY_ARRAY_STRUCTURE_AUTO.ARRAY_ARRAY_UINT[6][6];
    ARRAY_ARRAY_STRUCTURE_AUTO.ARRAY_ARRAY_UINT[7][7] := ARRAY_ARRAY_STRUCTURE_AUTO.ARRAY_ARRAY_UINT[6][7];
    ARRAY_ARRAY_STRUCTURE_AUTO.ARRAY_ARRAY_UINT[7][8] := ARRAY_ARRAY_STRUCTURE_AUTO.ARRAY_ARRAY_UINT[6][8];
    ARRAY_ARRAY_STRUCTURE_AUTO.ARRAY_ARRAY_UINT[7][9] := ARRAY_ARRAY_STRUCTURE_AUTO.ARRAY_ARRAY_UINT[6][9];

    ARRAY_ARRAY_STRUCTURE_AUTO.ARRAY_ARRAY_ULINT[0][0] := ARRAY_ARRAY_STRUCTURE_AUTO.ARRAY_ARRAY_ULINT[0][0] + 1;
    ARRAY_ARRAY_STRUCTURE_AUTO.ARRAY_ARRAY_ULINT[0][1] := ARRAY_ARRAY_STRUCTURE_AUTO.ARRAY_ARRAY_ULINT[0][1] + 1;
    ARRAY_ARRAY_STRUCTURE_AUTO.ARRAY_ARRAY_ULINT[0][2] := ARRAY_ARRAY_STRUCTURE_AUTO.ARRAY_ARRAY_ULINT[0][2] + 1;
    ARRAY_ARRAY_STRUCTURE_AUTO.ARRAY_ARRAY_ULINT[0][3] := ARRAY_ARRAY_STRUCTURE_AUTO.ARRAY_ARRAY_ULINT[0][3] + 1;
    ARRAY_ARRAY_STRUCTURE_AUTO.ARRAY_ARRAY_ULINT[0][4] := ARRAY_ARRAY_STRUCTURE_AUTO.ARRAY_ARRAY_ULINT[0][4] + 1;
    ARRAY_ARRAY_STRUCTURE_AUTO.ARRAY_ARRAY_ULINT[0][5] := ARRAY_ARRAY_STRUCTURE_AUTO.ARRAY_ARRAY_ULINT[0][5] + 1;
    ARRAY_ARRAY_STRUCTURE_AUTO.ARRAY_ARRAY_ULINT[0][6] := ARRAY_ARRAY_STRUCTURE_AUTO.ARRAY_ARRAY_ULINT[0][6] + 1;
    ARRAY_ARRAY_STRUCTURE_AUTO.ARRAY_ARRAY_ULINT[0][7] := ARRAY_ARRAY_STRUCTURE_AUTO.ARRAY_ARRAY_ULINT[0][7] + 1;
    ARRAY_ARRAY_STRUCTURE_AUTO.ARRAY_ARRAY_ULINT[0][8] := ARRAY_ARRAY_STRUCTURE_AUTO.ARRAY_ARRAY_ULINT[0][6];
    ARRAY_ARRAY_STRUCTURE_AUTO.ARRAY_ARRAY_ULINT[0][9] := ARRAY_ARRAY_STRUCTURE_AUTO.ARRAY_ARRAY_ULINT[0][7];

    ARRAY_ARRAY_STRUCTURE_AUTO.ARRAY_ARRAY_ULINT[1][0] := ARRAY_ARRAY_STRUCTURE_AUTO.ARRAY_ARRAY_ULINT[1][0] + 1;
    ARRAY_ARRAY_STRUCTURE_AUTO.ARRAY_ARRAY_ULINT[1][1] := ARRAY_ARRAY_STRUCTURE_AUTO.ARRAY_ARRAY_ULINT[1][1] + 1;
    ARRAY_ARRAY_STRUCTURE_AUTO.ARRAY_ARRAY_ULINT[1][2] := ARRAY_ARRAY_STRUCTURE_AUTO.ARRAY_ARRAY_ULINT[1][2] + 1;
    ARRAY_ARRAY_STRUCTURE_AUTO.ARRAY_ARRAY_ULINT[1][3] := ARRAY_ARRAY_STRUCTURE_AUTO.ARRAY_ARRAY_ULINT[1][3] + 1;
    ARRAY_ARRAY_STRUCTURE_AUTO.ARRAY_ARRAY_ULINT[1][4] := ARRAY_ARRAY_STRUCTURE_AUTO.ARRAY_ARRAY_ULINT[1][4] + 1;
    ARRAY_ARRAY_STRUCTURE_AUTO.ARRAY_ARRAY_ULINT[1][5] := ARRAY_ARRAY_STRUCTURE_AUTO.ARRAY_ARRAY_ULINT[1][5] + 1;
    ARRAY_ARRAY_STRUCTURE_AUTO.ARRAY_ARRAY_ULINT[1][6] := ARRAY_ARRAY_STRUCTURE_AUTO.ARRAY_ARRAY_ULINT[1][6] + 1;
    ARRAY_ARRAY_STRUCTURE_AUTO.ARRAY_ARRAY_ULINT[1][7] := ARRAY_ARRAY_STRUCTURE_AUTO.ARRAY_ARRAY_ULINT[1][7] + 1;
    ARRAY_ARRAY_STRUCTURE_AUTO.ARRAY_ARRAY_ULINT[1][8] := ARRAY_ARRAY_STRUCTURE_AUTO.ARRAY_ARRAY_ULINT[1][6];
    ARRAY_ARRAY_STRUCTURE_AUTO.ARRAY_ARRAY_ULINT[1][9] := ARRAY_ARRAY_STRUCTURE_AUTO.ARRAY_ARRAY_ULINT[1][7];

    ARRAY_ARRAY_STRUCTURE_AUTO.ARRAY_ARRAY_ULINT[2][0] := ARRAY_ARRAY_STRUCTURE_AUTO.ARRAY_ARRAY_ULINT[2][0] + 1;
    ARRAY_ARRAY_STRUCTURE_AUTO.ARRAY_ARRAY_ULINT[2][1] := ARRAY_ARRAY_STRUCTURE_AUTO.ARRAY_ARRAY_ULINT[2][1] + 1;
    ARRAY_ARRAY_STRUCTURE_AUTO.ARRAY_ARRAY_ULINT[2][2] := ARRAY_ARRAY_STRUCTURE_AUTO.ARRAY_ARRAY_ULINT[2][2] + 1;
    ARRAY_ARRAY_STRUCTURE_AUTO.ARRAY_ARRAY_ULINT[2][3] := ARRAY_ARRAY_STRUCTURE_AUTO.ARRAY_ARRAY_ULINT[2][3] + 1;
    ARRAY_ARRAY_STRUCTURE_AUTO.ARRAY_ARRAY_ULINT[2][4] := ARRAY_ARRAY_STRUCTURE_AUTO.ARRAY_ARRAY_ULINT[2][4] + 1;
    ARRAY_ARRAY_STRUCTURE_AUTO.ARRAY_ARRAY_ULINT[2][5] := ARRAY_ARRAY_STRUCTURE_AUTO.ARRAY_ARRAY_ULINT[2][5] + 1;
    ARRAY_ARRAY_STRUCTURE_AUTO.ARRAY_ARRAY_ULINT[2][6] := ARRAY_ARRAY_STRUCTURE_AUTO.ARRAY_ARRAY_ULINT[2][6] + 1;
    ARRAY_ARRAY_STRUCTURE_AUTO.ARRAY_ARRAY_ULINT[2][7] := ARRAY_ARRAY_STRUCTURE_AUTO.ARRAY_ARRAY_ULINT[2][7] + 1;
    ARRAY_ARRAY_STRUCTURE_AUTO.ARRAY_ARRAY_ULINT[2][8] := ARRAY_ARRAY_STRUCTURE_AUTO.ARRAY_ARRAY_ULINT[2][8] + 1;
    ARRAY_ARRAY_STRUCTURE_AUTO.ARRAY_ARRAY_ULINT[2][9] := ARRAY_ARRAY_STRUCTURE_AUTO.ARRAY_ARRAY_ULINT[2][9] + 1;

    ARRAY_ARRAY_STRUCTURE_AUTO.ARRAY_ARRAY_ULINT[3][0] := ARRAY_ARRAY_STRUCTURE_AUTO.ARRAY_ARRAY_ULINT[3][0] + 1;
    ARRAY_ARRAY_STRUCTURE_AUTO.ARRAY_ARRAY_ULINT[3][1] := ARRAY_ARRAY_STRUCTURE_AUTO.ARRAY_ARRAY_ULINT[3][1] + 1;
    ARRAY_ARRAY_STRUCTURE_AUTO.ARRAY_ARRAY_ULINT[3][2] := ARRAY_ARRAY_STRUCTURE_AUTO.ARRAY_ARRAY_ULINT[3][2] + 1;
    ARRAY_ARRAY_STRUCTURE_AUTO.ARRAY_ARRAY_ULINT[3][3] := ARRAY_ARRAY_STRUCTURE_AUTO.ARRAY_ARRAY_ULINT[3][3] + 1;
    ARRAY_ARRAY_STRUCTURE_AUTO.ARRAY_ARRAY_ULINT[3][4] := ARRAY_ARRAY_STRUCTURE_AUTO.ARRAY_ARRAY_ULINT[3][4] + 1;
    ARRAY_ARRAY_STRUCTURE_AUTO.ARRAY_ARRAY_ULINT[3][5] := ARRAY_ARRAY_STRUCTURE_AUTO.ARRAY_ARRAY_ULINT[3][5] + 1;
    ARRAY_ARRAY_STRUCTURE_AUTO.ARRAY_ARRAY_ULINT[3][6] := ARRAY_ARRAY_STRUCTURE_AUTO.ARRAY_ARRAY_ULINT[3][6] + 1;
    ARRAY_ARRAY_STRUCTURE_AUTO.ARRAY_ARRAY_ULINT[3][7] := ARRAY_ARRAY_STRUCTURE_AUTO.ARRAY_ARRAY_ULINT[3][7] + 1;
    ARRAY_ARRAY_STRUCTURE_AUTO.ARRAY_ARRAY_ULINT[3][8] := ARRAY_ARRAY_STRUCTURE_AUTO.ARRAY_ARRAY_ULINT[3][8] + 1;
    ARRAY_ARRAY_STRUCTURE_AUTO.ARRAY_ARRAY_ULINT[3][9] := ARRAY_ARRAY_STRUCTURE_AUTO.ARRAY_ARRAY_ULINT[3][8] + 1;

    ARRAY_ARRAY_STRUCTURE_AUTO.ARRAY_ARRAY_ULINT[4][0] := ARRAY_ARRAY_STRUCTURE_AUTO.ARRAY_ARRAY_ULINT[4][0] + 1;
    ARRAY_ARRAY_STRUCTURE_AUTO.ARRAY_ARRAY_ULINT[4][1] := ARRAY_ARRAY_STRUCTURE_AUTO.ARRAY_ARRAY_ULINT[4][1] + 1;
    ARRAY_ARRAY_STRUCTURE_AUTO.ARRAY_ARRAY_ULINT[4][2] := ARRAY_ARRAY_STRUCTURE_AUTO.ARRAY_ARRAY_ULINT[4][2] + 1;
    ARRAY_ARRAY_STRUCTURE_AUTO.ARRAY_ARRAY_ULINT[4][3] := ARRAY_ARRAY_STRUCTURE_AUTO.ARRAY_ARRAY_ULINT[4][3] + 1;
    ARRAY_ARRAY_STRUCTURE_AUTO.ARRAY_ARRAY_ULINT[4][4] := ARRAY_ARRAY_STRUCTURE_AUTO.ARRAY_ARRAY_ULINT[4][4] + 1;
    ARRAY_ARRAY_STRUCTURE_AUTO.ARRAY_ARRAY_ULINT[4][5] := ARRAY_ARRAY_STRUCTURE_AUTO.ARRAY_ARRAY_ULINT[4][5] + 1;
    ARRAY_ARRAY_STRUCTURE_AUTO.ARRAY_ARRAY_ULINT[4][6] := ARRAY_ARRAY_STRUCTURE_AUTO.ARRAY_ARRAY_ULINT[4][6] + 1;
    ARRAY_ARRAY_STRUCTURE_AUTO.ARRAY_ARRAY_ULINT[4][7] := ARRAY_ARRAY_STRUCTURE_AUTO.ARRAY_ARRAY_ULINT[4][7] + 1;
    ARRAY_ARRAY_STRUCTURE_AUTO.ARRAY_ARRAY_ULINT[4][8] := ARRAY_ARRAY_STRUCTURE_AUTO.ARRAY_ARRAY_ULINT[4][8] + 1;
    ARRAY_ARRAY_STRUCTURE_AUTO.ARRAY_ARRAY_ULINT[4][9] := ARRAY_ARRAY_STRUCTURE_AUTO.ARRAY_ARRAY_ULINT[4][9] + 1;

    ARRAY_ARRAY_STRUCTURE_AUTO.ARRAY_ARRAY_ULINT[5][0] := ARRAY_ARRAY_STRUCTURE_AUTO.ARRAY_ARRAY_ULINT[5][0] + 1;
    ARRAY_ARRAY_STRUCTURE_AUTO.ARRAY_ARRAY_ULINT[5][1] := ARRAY_ARRAY_STRUCTURE_AUTO.ARRAY_ARRAY_ULINT[5][1] + 1;
    ARRAY_ARRAY_STRUCTURE_AUTO.ARRAY_ARRAY_ULINT[5][2] := ARRAY_ARRAY_STRUCTURE_AUTO.ARRAY_ARRAY_ULINT[5][2] + 1;
    ARRAY_ARRAY_STRUCTURE_AUTO.ARRAY_ARRAY_ULINT[5][3] := ARRAY_ARRAY_STRUCTURE_AUTO.ARRAY_ARRAY_ULINT[5][3] + 1;
    ARRAY_ARRAY_STRUCTURE_AUTO.ARRAY_ARRAY_ULINT[5][4] := ARRAY_ARRAY_STRUCTURE_AUTO.ARRAY_ARRAY_ULINT[5][4] + 1;
    ARRAY_ARRAY_STRUCTURE_AUTO.ARRAY_ARRAY_ULINT[5][5] := ARRAY_ARRAY_STRUCTURE_AUTO.ARRAY_ARRAY_ULINT[5][5] + 1;
    ARRAY_ARRAY_STRUCTURE_AUTO.ARRAY_ARRAY_ULINT[5][6] := ARRAY_ARRAY_STRUCTURE_AUTO.ARRAY_ARRAY_ULINT[5][6] + 1;
    ARRAY_ARRAY_STRUCTURE_AUTO.ARRAY_ARRAY_ULINT[5][7] := ARRAY_ARRAY_STRUCTURE_AUTO.ARRAY_ARRAY_ULINT[5][7] + 1;
    ARRAY_ARRAY_STRUCTURE_AUTO.ARRAY_ARRAY_ULINT[5][8] := ARRAY_ARRAY_STRUCTURE_AUTO.ARRAY_ARRAY_ULINT[5][8] + 1;
    ARRAY_ARRAY_STRUCTURE_AUTO.ARRAY_ARRAY_ULINT[5][9] := ARRAY_ARRAY_STRUCTURE_AUTO.ARRAY_ARRAY_ULINT[5][9] + 1;

    ARRAY_ARRAY_STRUCTURE_AUTO.ARRAY_ARRAY_ULINT[6][0] := ARRAY_ARRAY_STRUCTURE_AUTO.ARRAY_ARRAY_ULINT[6][0] + 1;
    ARRAY_ARRAY_STRUCTURE_AUTO.ARRAY_ARRAY_ULINT[6][1] := ARRAY_ARRAY_STRUCTURE_AUTO.ARRAY_ARRAY_ULINT[6][1] + 1;
    ARRAY_ARRAY_STRUCTURE_AUTO.ARRAY_ARRAY_ULINT[6][2] := ARRAY_ARRAY_STRUCTURE_AUTO.ARRAY_ARRAY_ULINT[6][2] + 1;
    ARRAY_ARRAY_STRUCTURE_AUTO.ARRAY_ARRAY_ULINT[6][3] := ARRAY_ARRAY_STRUCTURE_AUTO.ARRAY_ARRAY_ULINT[6][3] + 1;
    ARRAY_ARRAY_STRUCTURE_AUTO.ARRAY_ARRAY_ULINT[6][4] := ARRAY_ARRAY_STRUCTURE_AUTO.ARRAY_ARRAY_ULINT[6][4] + 1;
    ARRAY_ARRAY_STRUCTURE_AUTO.ARRAY_ARRAY_ULINT[6][5] := ARRAY_ARRAY_STRUCTURE_AUTO.ARRAY_ARRAY_ULINT[6][5] + 1;
    ARRAY_ARRAY_STRUCTURE_AUTO.ARRAY_ARRAY_ULINT[6][6] := ARRAY_ARRAY_STRUCTURE_AUTO.ARRAY_ARRAY_ULINT[6][6] + 1;
    ARRAY_ARRAY_STRUCTURE_AUTO.ARRAY_ARRAY_ULINT[6][7] := ARRAY_ARRAY_STRUCTURE_AUTO.ARRAY_ARRAY_ULINT[6][7] + 1;
    ARRAY_ARRAY_STRUCTURE_AUTO.ARRAY_ARRAY_ULINT[6][8] := ARRAY_ARRAY_STRUCTURE_AUTO.ARRAY_ARRAY_ULINT[6][8] + 1;
    ARRAY_ARRAY_STRUCTURE_AUTO.ARRAY_ARRAY_ULINT[6][9] := ARRAY_ARRAY_STRUCTURE_AUTO.ARRAY_ARRAY_ULINT[6][9] + 1;

    ARRAY_ARRAY_STRUCTURE_AUTO.ARRAY_ARRAY_ULINT[7][0] := ARRAY_ARRAY_STRUCTURE_AUTO.ARRAY_ARRAY_ULINT[6][0];
    ARRAY_ARRAY_STRUCTURE_AUTO.ARRAY_ARRAY_ULINT[7][1] := ARRAY_ARRAY_STRUCTURE_AUTO.ARRAY_ARRAY_ULINT[6][1];
    ARRAY_ARRAY_STRUCTURE_AUTO.ARRAY_ARRAY_ULINT[7][2] := ARRAY_ARRAY_STRUCTURE_AUTO.ARRAY_ARRAY_ULINT[6][2];
    ARRAY_ARRAY_STRUCTURE_AUTO.ARRAY_ARRAY_ULINT[7][3] := ARRAY_ARRAY_STRUCTURE_AUTO.ARRAY_ARRAY_ULINT[6][3];
    ARRAY_ARRAY_STRUCTURE_AUTO.ARRAY_ARRAY_ULINT[7][4] := ARRAY_ARRAY_STRUCTURE_AUTO.ARRAY_ARRAY_ULINT[6][4];
    ARRAY_ARRAY_STRUCTURE_AUTO.ARRAY_ARRAY_ULINT[7][5] := ARRAY_ARRAY_STRUCTURE_AUTO.ARRAY_ARRAY_ULINT[6][5];
    ARRAY_ARRAY_STRUCTURE_AUTO.ARRAY_ARRAY_ULINT[7][6] := ARRAY_ARRAY_STRUCTURE_AUTO.ARRAY_ARRAY_ULINT[6][6];
    ARRAY_ARRAY_STRUCTURE_AUTO.ARRAY_ARRAY_ULINT[7][7] := ARRAY_ARRAY_STRUCTURE_AUTO.ARRAY_ARRAY_ULINT[6][7];
    ARRAY_ARRAY_STRUCTURE_AUTO.ARRAY_ARRAY_ULINT[7][8] := ARRAY_ARRAY_STRUCTURE_AUTO.ARRAY_ARRAY_ULINT[6][8];
    ARRAY_ARRAY_STRUCTURE_AUTO.ARRAY_ARRAY_ULINT[7][9] := ARRAY_ARRAY_STRUCTURE_AUTO.ARRAY_ARRAY_ULINT[6][9];

    ARRAY_ARRAY_STRUCTURE_AUTO.ARRAY_ARRAY_USINT[0][0] := ARRAY_ARRAY_STRUCTURE_AUTO.ARRAY_ARRAY_USINT[0][0] + 1;
    ARRAY_ARRAY_STRUCTURE_AUTO.ARRAY_ARRAY_USINT[0][1] := ARRAY_ARRAY_STRUCTURE_AUTO.ARRAY_ARRAY_USINT[0][1] + 1;
    ARRAY_ARRAY_STRUCTURE_AUTO.ARRAY_ARRAY_USINT[0][2] := ARRAY_ARRAY_STRUCTURE_AUTO.ARRAY_ARRAY_USINT[0][2] + 1;
    ARRAY_ARRAY_STRUCTURE_AUTO.ARRAY_ARRAY_USINT[0][3] := ARRAY_ARRAY_STRUCTURE_AUTO.ARRAY_ARRAY_USINT[0][3] + 1;
    ARRAY_ARRAY_STRUCTURE_AUTO.ARRAY_ARRAY_USINT[0][4] := ARRAY_ARRAY_STRUCTURE_AUTO.ARRAY_ARRAY_USINT[0][4] + 1;
    ARRAY_ARRAY_STRUCTURE_AUTO.ARRAY_ARRAY_USINT[0][5] := ARRAY_ARRAY_STRUCTURE_AUTO.ARRAY_ARRAY_USINT[0][5] + 1;
    ARRAY_ARRAY_STRUCTURE_AUTO.ARRAY_ARRAY_USINT[0][6] := ARRAY_ARRAY_STRUCTURE_AUTO.ARRAY_ARRAY_USINT[0][6] + 1;
    ARRAY_ARRAY_STRUCTURE_AUTO.ARRAY_ARRAY_USINT[0][7] := ARRAY_ARRAY_STRUCTURE_AUTO.ARRAY_ARRAY_USINT[0][7] + 1;
    ARRAY_ARRAY_STRUCTURE_AUTO.ARRAY_ARRAY_USINT[0][8] := ARRAY_ARRAY_STRUCTURE_AUTO.ARRAY_ARRAY_USINT[0][6];
    ARRAY_ARRAY_STRUCTURE_AUTO.ARRAY_ARRAY_USINT[0][9] := ARRAY_ARRAY_STRUCTURE_AUTO.ARRAY_ARRAY_USINT[0][7];

    ARRAY_ARRAY_STRUCTURE_AUTO.ARRAY_ARRAY_USINT[1][0] := ARRAY_ARRAY_STRUCTURE_AUTO.ARRAY_ARRAY_USINT[1][0] + 1;
    ARRAY_ARRAY_STRUCTURE_AUTO.ARRAY_ARRAY_USINT[1][1] := ARRAY_ARRAY_STRUCTURE_AUTO.ARRAY_ARRAY_USINT[1][1] + 1;
    ARRAY_ARRAY_STRUCTURE_AUTO.ARRAY_ARRAY_USINT[1][2] := ARRAY_ARRAY_STRUCTURE_AUTO.ARRAY_ARRAY_USINT[1][2] + 1;
    ARRAY_ARRAY_STRUCTURE_AUTO.ARRAY_ARRAY_USINT[1][3] := ARRAY_ARRAY_STRUCTURE_AUTO.ARRAY_ARRAY_USINT[1][3] + 1;
    ARRAY_ARRAY_STRUCTURE_AUTO.ARRAY_ARRAY_USINT[1][4] := ARRAY_ARRAY_STRUCTURE_AUTO.ARRAY_ARRAY_USINT[1][4] + 1;
    ARRAY_ARRAY_STRUCTURE_AUTO.ARRAY_ARRAY_USINT[1][5] := ARRAY_ARRAY_STRUCTURE_AUTO.ARRAY_ARRAY_USINT[1][5] + 1;
    ARRAY_ARRAY_STRUCTURE_AUTO.ARRAY_ARRAY_USINT[1][6] := ARRAY_ARRAY_STRUCTURE_AUTO.ARRAY_ARRAY_USINT[1][6] + 1;
    ARRAY_ARRAY_STRUCTURE_AUTO.ARRAY_ARRAY_USINT[1][7] := ARRAY_ARRAY_STRUCTURE_AUTO.ARRAY_ARRAY_USINT[1][7] + 1;
    ARRAY_ARRAY_STRUCTURE_AUTO.ARRAY_ARRAY_USINT[1][8] := ARRAY_ARRAY_STRUCTURE_AUTO.ARRAY_ARRAY_USINT[1][6];
    ARRAY_ARRAY_STRUCTURE_AUTO.ARRAY_ARRAY_USINT[1][9] := ARRAY_ARRAY_STRUCTURE_AUTO.ARRAY_ARRAY_USINT[1][7];

    ARRAY_ARRAY_STRUCTURE_AUTO.ARRAY_ARRAY_USINT[2][0] := ARRAY_ARRAY_STRUCTURE_AUTO.ARRAY_ARRAY_USINT[2][0] + 1;
    ARRAY_ARRAY_STRUCTURE_AUTO.ARRAY_ARRAY_USINT[2][1] := ARRAY_ARRAY_STRUCTURE_AUTO.ARRAY_ARRAY_USINT[2][1] + 1;
    ARRAY_ARRAY_STRUCTURE_AUTO.ARRAY_ARRAY_USINT[2][2] := ARRAY_ARRAY_STRUCTURE_AUTO.ARRAY_ARRAY_USINT[2][2] + 1;
    ARRAY_ARRAY_STRUCTURE_AUTO.ARRAY_ARRAY_USINT[2][3] := ARRAY_ARRAY_STRUCTURE_AUTO.ARRAY_ARRAY_USINT[2][3] + 1;
    ARRAY_ARRAY_STRUCTURE_AUTO.ARRAY_ARRAY_USINT[2][4] := ARRAY_ARRAY_STRUCTURE_AUTO.ARRAY_ARRAY_USINT[2][4] + 1;
    ARRAY_ARRAY_STRUCTURE_AUTO.ARRAY_ARRAY_USINT[2][5] := ARRAY_ARRAY_STRUCTURE_AUTO.ARRAY_ARRAY_USINT[2][5] + 1;
    ARRAY_ARRAY_STRUCTURE_AUTO.ARRAY_ARRAY_USINT[2][6] := ARRAY_ARRAY_STRUCTURE_AUTO.ARRAY_ARRAY_USINT[2][6] + 1;
    ARRAY_ARRAY_STRUCTURE_AUTO.ARRAY_ARRAY_USINT[2][7] := ARRAY_ARRAY_STRUCTURE_AUTO.ARRAY_ARRAY_USINT[2][7] + 1;
    ARRAY_ARRAY_STRUCTURE_AUTO.ARRAY_ARRAY_USINT[2][8] := ARRAY_ARRAY_STRUCTURE_AUTO.ARRAY_ARRAY_USINT[2][8] + 1;
    ARRAY_ARRAY_STRUCTURE_AUTO.ARRAY_ARRAY_USINT[2][9] := ARRAY_ARRAY_STRUCTURE_AUTO.ARRAY_ARRAY_USINT[2][9] + 1;

    ARRAY_ARRAY_STRUCTURE_AUTO.ARRAY_ARRAY_USINT[3][0] := ARRAY_ARRAY_STRUCTURE_AUTO.ARRAY_ARRAY_USINT[3][0] + 1;
    ARRAY_ARRAY_STRUCTURE_AUTO.ARRAY_ARRAY_USINT[3][1] := ARRAY_ARRAY_STRUCTURE_AUTO.ARRAY_ARRAY_USINT[3][1] + 1;
    ARRAY_ARRAY_STRUCTURE_AUTO.ARRAY_ARRAY_USINT[3][2] := ARRAY_ARRAY_STRUCTURE_AUTO.ARRAY_ARRAY_USINT[3][2] + 1;
    ARRAY_ARRAY_STRUCTURE_AUTO.ARRAY_ARRAY_USINT[3][3] := ARRAY_ARRAY_STRUCTURE_AUTO.ARRAY_ARRAY_USINT[3][3] + 1;
    ARRAY_ARRAY_STRUCTURE_AUTO.ARRAY_ARRAY_USINT[3][4] := ARRAY_ARRAY_STRUCTURE_AUTO.ARRAY_ARRAY_USINT[3][4] + 1;
    ARRAY_ARRAY_STRUCTURE_AUTO.ARRAY_ARRAY_USINT[3][5] := ARRAY_ARRAY_STRUCTURE_AUTO.ARRAY_ARRAY_USINT[3][5] + 1;
    ARRAY_ARRAY_STRUCTURE_AUTO.ARRAY_ARRAY_USINT[3][6] := ARRAY_ARRAY_STRUCTURE_AUTO.ARRAY_ARRAY_USINT[3][6] + 1;
    ARRAY_ARRAY_STRUCTURE_AUTO.ARRAY_ARRAY_USINT[3][7] := ARRAY_ARRAY_STRUCTURE_AUTO.ARRAY_ARRAY_USINT[3][7] + 1;
    ARRAY_ARRAY_STRUCTURE_AUTO.ARRAY_ARRAY_USINT[3][8] := ARRAY_ARRAY_STRUCTURE_AUTO.ARRAY_ARRAY_USINT[3][8] + 1;
    ARRAY_ARRAY_STRUCTURE_AUTO.ARRAY_ARRAY_USINT[3][9] := ARRAY_ARRAY_STRUCTURE_AUTO.ARRAY_ARRAY_USINT[3][8] + 1;

    ARRAY_ARRAY_STRUCTURE_AUTO.ARRAY_ARRAY_USINT[4][0] := ARRAY_ARRAY_STRUCTURE_AUTO.ARRAY_ARRAY_USINT[4][0] + 1;
    ARRAY_ARRAY_STRUCTURE_AUTO.ARRAY_ARRAY_USINT[4][1] := ARRAY_ARRAY_STRUCTURE_AUTO.ARRAY_ARRAY_USINT[4][1] + 1;
    ARRAY_ARRAY_STRUCTURE_AUTO.ARRAY_ARRAY_USINT[4][2] := ARRAY_ARRAY_STRUCTURE_AUTO.ARRAY_ARRAY_USINT[4][2] + 1;
    ARRAY_ARRAY_STRUCTURE_AUTO.ARRAY_ARRAY_USINT[4][3] := ARRAY_ARRAY_STRUCTURE_AUTO.ARRAY_ARRAY_USINT[4][3] + 1;
    ARRAY_ARRAY_STRUCTURE_AUTO.ARRAY_ARRAY_USINT[4][4] := ARRAY_ARRAY_STRUCTURE_AUTO.ARRAY_ARRAY_USINT[4][4] + 1;
    ARRAY_ARRAY_STRUCTURE_AUTO.ARRAY_ARRAY_USINT[4][5] := ARRAY_ARRAY_STRUCTURE_AUTO.ARRAY_ARRAY_USINT[4][5] + 1;
    ARRAY_ARRAY_STRUCTURE_AUTO.ARRAY_ARRAY_USINT[4][6] := ARRAY_ARRAY_STRUCTURE_AUTO.ARRAY_ARRAY_USINT[4][6] + 1;
    ARRAY_ARRAY_STRUCTURE_AUTO.ARRAY_ARRAY_USINT[4][7] := ARRAY_ARRAY_STRUCTURE_AUTO.ARRAY_ARRAY_USINT[4][7] + 1;
    ARRAY_ARRAY_STRUCTURE_AUTO.ARRAY_ARRAY_USINT[4][8] := ARRAY_ARRAY_STRUCTURE_AUTO.ARRAY_ARRAY_USINT[4][8] + 1;
    ARRAY_ARRAY_STRUCTURE_AUTO.ARRAY_ARRAY_USINT[4][9] := ARRAY_ARRAY_STRUCTURE_AUTO.ARRAY_ARRAY_USINT[4][9] + 1;

    ARRAY_ARRAY_STRUCTURE_AUTO.ARRAY_ARRAY_USINT[5][0] := ARRAY_ARRAY_STRUCTURE_AUTO.ARRAY_ARRAY_USINT[5][0] + 1;
    ARRAY_ARRAY_STRUCTURE_AUTO.ARRAY_ARRAY_USINT[5][1] := ARRAY_ARRAY_STRUCTURE_AUTO.ARRAY_ARRAY_USINT[5][1] + 1;
    ARRAY_ARRAY_STRUCTURE_AUTO.ARRAY_ARRAY_USINT[5][2] := ARRAY_ARRAY_STRUCTURE_AUTO.ARRAY_ARRAY_USINT[5][2] + 1;
    ARRAY_ARRAY_STRUCTURE_AUTO.ARRAY_ARRAY_USINT[5][3] := ARRAY_ARRAY_STRUCTURE_AUTO.ARRAY_ARRAY_USINT[5][3] + 1;
    ARRAY_ARRAY_STRUCTURE_AUTO.ARRAY_ARRAY_USINT[5][4] := ARRAY_ARRAY_STRUCTURE_AUTO.ARRAY_ARRAY_USINT[5][4] + 1;
    ARRAY_ARRAY_STRUCTURE_AUTO.ARRAY_ARRAY_USINT[5][5] := ARRAY_ARRAY_STRUCTURE_AUTO.ARRAY_ARRAY_USINT[5][5] + 1;
    ARRAY_ARRAY_STRUCTURE_AUTO.ARRAY_ARRAY_USINT[5][6] := ARRAY_ARRAY_STRUCTURE_AUTO.ARRAY_ARRAY_USINT[5][6] + 1;
    ARRAY_ARRAY_STRUCTURE_AUTO.ARRAY_ARRAY_USINT[5][7] := ARRAY_ARRAY_STRUCTURE_AUTO.ARRAY_ARRAY_USINT[5][7] + 1;
    ARRAY_ARRAY_STRUCTURE_AUTO.ARRAY_ARRAY_USINT[5][8] := ARRAY_ARRAY_STRUCTURE_AUTO.ARRAY_ARRAY_USINT[5][8] + 1;
    ARRAY_ARRAY_STRUCTURE_AUTO.ARRAY_ARRAY_USINT[5][9] := ARRAY_ARRAY_STRUCTURE_AUTO.ARRAY_ARRAY_USINT[5][9] + 1;

    ARRAY_ARRAY_STRUCTURE_AUTO.ARRAY_ARRAY_USINT[6][0] := ARRAY_ARRAY_STRUCTURE_AUTO.ARRAY_ARRAY_USINT[6][0] + 1;
    ARRAY_ARRAY_STRUCTURE_AUTO.ARRAY_ARRAY_USINT[6][1] := ARRAY_ARRAY_STRUCTURE_AUTO.ARRAY_ARRAY_USINT[6][1] + 1;
    ARRAY_ARRAY_STRUCTURE_AUTO.ARRAY_ARRAY_USINT[6][2] := ARRAY_ARRAY_STRUCTURE_AUTO.ARRAY_ARRAY_USINT[6][2] + 1;
    ARRAY_ARRAY_STRUCTURE_AUTO.ARRAY_ARRAY_USINT[6][3] := ARRAY_ARRAY_STRUCTURE_AUTO.ARRAY_ARRAY_USINT[6][3] + 1;
    ARRAY_ARRAY_STRUCTURE_AUTO.ARRAY_ARRAY_USINT[6][4] := ARRAY_ARRAY_STRUCTURE_AUTO.ARRAY_ARRAY_USINT[6][4] + 1;
    ARRAY_ARRAY_STRUCTURE_AUTO.ARRAY_ARRAY_USINT[6][5] := ARRAY_ARRAY_STRUCTURE_AUTO.ARRAY_ARRAY_USINT[6][5] + 1;
    ARRAY_ARRAY_STRUCTURE_AUTO.ARRAY_ARRAY_USINT[6][6] := ARRAY_ARRAY_STRUCTURE_AUTO.ARRAY_ARRAY_USINT[6][6] + 1;
    ARRAY_ARRAY_STRUCTURE_AUTO.ARRAY_ARRAY_USINT[6][7] := ARRAY_ARRAY_STRUCTURE_AUTO.ARRAY_ARRAY_USINT[6][7] + 1;
    ARRAY_ARRAY_STRUCTURE_AUTO.ARRAY_ARRAY_USINT[6][8] := ARRAY_ARRAY_STRUCTURE_AUTO.ARRAY_ARRAY_USINT[6][8] + 1;
    ARRAY_ARRAY_STRUCTURE_AUTO.ARRAY_ARRAY_USINT[6][9] := ARRAY_ARRAY_STRUCTURE_AUTO.ARRAY_ARRAY_USINT[6][9] + 1;

    ARRAY_ARRAY_STRUCTURE_AUTO.ARRAY_ARRAY_USINT[7][0] := ARRAY_ARRAY_STRUCTURE_AUTO.ARRAY_ARRAY_USINT[6][0];
    ARRAY_ARRAY_STRUCTURE_AUTO.ARRAY_ARRAY_USINT[7][1] := ARRAY_ARRAY_STRUCTURE_AUTO.ARRAY_ARRAY_USINT[6][1];
    ARRAY_ARRAY_STRUCTURE_AUTO.ARRAY_ARRAY_USINT[7][2] := ARRAY_ARRAY_STRUCTURE_AUTO.ARRAY_ARRAY_USINT[6][2];
    ARRAY_ARRAY_STRUCTURE_AUTO.ARRAY_ARRAY_USINT[7][3] := ARRAY_ARRAY_STRUCTURE_AUTO.ARRAY_ARRAY_USINT[6][3];
    ARRAY_ARRAY_STRUCTURE_AUTO.ARRAY_ARRAY_USINT[7][4] := ARRAY_ARRAY_STRUCTURE_AUTO.ARRAY_ARRAY_USINT[6][4];
    ARRAY_ARRAY_STRUCTURE_AUTO.ARRAY_ARRAY_USINT[7][5] := ARRAY_ARRAY_STRUCTURE_AUTO.ARRAY_ARRAY_USINT[6][5];
    ARRAY_ARRAY_STRUCTURE_AUTO.ARRAY_ARRAY_USINT[7][6] := ARRAY_ARRAY_STRUCTURE_AUTO.ARRAY_ARRAY_USINT[6][6];
    ARRAY_ARRAY_STRUCTURE_AUTO.ARRAY_ARRAY_USINT[7][7] := ARRAY_ARRAY_STRUCTURE_AUTO.ARRAY_ARRAY_USINT[6][7];
    ARRAY_ARRAY_STRUCTURE_AUTO.ARRAY_ARRAY_USINT[7][8] := ARRAY_ARRAY_STRUCTURE_AUTO.ARRAY_ARRAY_USINT[6][8];
    ARRAY_ARRAY_STRUCTURE_AUTO.ARRAY_ARRAY_USINT[7][9] := ARRAY_ARRAY_STRUCTURE_AUTO.ARRAY_ARRAY_USINT[6][9];

    ARRAY_ARRAY_STRUCTURE_AUTO.ARRAY_ARRAY_WORD[0][0] := ARRAY_ARRAY_STRUCTURE_AUTO.ARRAY_ARRAY_WORD[0][0] + 1;
    ARRAY_ARRAY_STRUCTURE_AUTO.ARRAY_ARRAY_WORD[0][1] := ARRAY_ARRAY_STRUCTURE_AUTO.ARRAY_ARRAY_WORD[0][1] + 1;
    ARRAY_ARRAY_STRUCTURE_AUTO.ARRAY_ARRAY_WORD[0][2] := ARRAY_ARRAY_STRUCTURE_AUTO.ARRAY_ARRAY_WORD[0][2] + 1;
    ARRAY_ARRAY_STRUCTURE_AUTO.ARRAY_ARRAY_WORD[0][3] := ARRAY_ARRAY_STRUCTURE_AUTO.ARRAY_ARRAY_WORD[0][3] + 1;
    ARRAY_ARRAY_STRUCTURE_AUTO.ARRAY_ARRAY_WORD[0][4] := ARRAY_ARRAY_STRUCTURE_AUTO.ARRAY_ARRAY_WORD[0][4] + 1;
    ARRAY_ARRAY_STRUCTURE_AUTO.ARRAY_ARRAY_WORD[0][5] := ARRAY_ARRAY_STRUCTURE_AUTO.ARRAY_ARRAY_WORD[0][5] + 1;
    ARRAY_ARRAY_STRUCTURE_AUTO.ARRAY_ARRAY_WORD[0][6] := ARRAY_ARRAY_STRUCTURE_AUTO.ARRAY_ARRAY_WORD[0][6] + 1;
    ARRAY_ARRAY_STRUCTURE_AUTO.ARRAY_ARRAY_WORD[0][7] := ARRAY_ARRAY_STRUCTURE_AUTO.ARRAY_ARRAY_WORD[0][7] + 1;
    ARRAY_ARRAY_STRUCTURE_AUTO.ARRAY_ARRAY_WORD[0][8] := ARRAY_ARRAY_STRUCTURE_AUTO.ARRAY_ARRAY_WORD[0][6];
    ARRAY_ARRAY_STRUCTURE_AUTO.ARRAY_ARRAY_WORD[0][9] := ARRAY_ARRAY_STRUCTURE_AUTO.ARRAY_ARRAY_WORD[0][7];

    ARRAY_ARRAY_STRUCTURE_AUTO.ARRAY_ARRAY_WORD[1][0] := ARRAY_ARRAY_STRUCTURE_AUTO.ARRAY_ARRAY_WORD[1][0] + 1;
    ARRAY_ARRAY_STRUCTURE_AUTO.ARRAY_ARRAY_WORD[1][1] := ARRAY_ARRAY_STRUCTURE_AUTO.ARRAY_ARRAY_WORD[1][1] + 1;
    ARRAY_ARRAY_STRUCTURE_AUTO.ARRAY_ARRAY_WORD[1][2] := ARRAY_ARRAY_STRUCTURE_AUTO.ARRAY_ARRAY_WORD[1][2] + 1;
    ARRAY_ARRAY_STRUCTURE_AUTO.ARRAY_ARRAY_WORD[1][3] := ARRAY_ARRAY_STRUCTURE_AUTO.ARRAY_ARRAY_WORD[1][3] + 1;
    ARRAY_ARRAY_STRUCTURE_AUTO.ARRAY_ARRAY_WORD[1][4] := ARRAY_ARRAY_STRUCTURE_AUTO.ARRAY_ARRAY_WORD[1][4] + 1;
    ARRAY_ARRAY_STRUCTURE_AUTO.ARRAY_ARRAY_WORD[1][5] := ARRAY_ARRAY_STRUCTURE_AUTO.ARRAY_ARRAY_WORD[1][5] + 1;
    ARRAY_ARRAY_STRUCTURE_AUTO.ARRAY_ARRAY_WORD[1][6] := ARRAY_ARRAY_STRUCTURE_AUTO.ARRAY_ARRAY_WORD[1][6] + 1;
    ARRAY_ARRAY_STRUCTURE_AUTO.ARRAY_ARRAY_WORD[1][7] := ARRAY_ARRAY_STRUCTURE_AUTO.ARRAY_ARRAY_WORD[1][7] + 1;
    ARRAY_ARRAY_STRUCTURE_AUTO.ARRAY_ARRAY_WORD[1][8] := ARRAY_ARRAY_STRUCTURE_AUTO.ARRAY_ARRAY_WORD[1][6];
    ARRAY_ARRAY_STRUCTURE_AUTO.ARRAY_ARRAY_WORD[1][9] := ARRAY_ARRAY_STRUCTURE_AUTO.ARRAY_ARRAY_WORD[1][7];

    ARRAY_ARRAY_STRUCTURE_AUTO.ARRAY_ARRAY_WORD[2][0] := ARRAY_ARRAY_STRUCTURE_AUTO.ARRAY_ARRAY_WORD[2][0] + 1;
    ARRAY_ARRAY_STRUCTURE_AUTO.ARRAY_ARRAY_WORD[2][1] := ARRAY_ARRAY_STRUCTURE_AUTO.ARRAY_ARRAY_WORD[2][1] + 1;
    ARRAY_ARRAY_STRUCTURE_AUTO.ARRAY_ARRAY_WORD[2][2] := ARRAY_ARRAY_STRUCTURE_AUTO.ARRAY_ARRAY_WORD[2][2] + 1;
    ARRAY_ARRAY_STRUCTURE_AUTO.ARRAY_ARRAY_WORD[2][3] := ARRAY_ARRAY_STRUCTURE_AUTO.ARRAY_ARRAY_WORD[2][3] + 1;
    ARRAY_ARRAY_STRUCTURE_AUTO.ARRAY_ARRAY_WORD[2][4] := ARRAY_ARRAY_STRUCTURE_AUTO.ARRAY_ARRAY_WORD[2][4] + 1;
    ARRAY_ARRAY_STRUCTURE_AUTO.ARRAY_ARRAY_WORD[2][5] := ARRAY_ARRAY_STRUCTURE_AUTO.ARRAY_ARRAY_WORD[2][5] + 1;
    ARRAY_ARRAY_STRUCTURE_AUTO.ARRAY_ARRAY_WORD[2][6] := ARRAY_ARRAY_STRUCTURE_AUTO.ARRAY_ARRAY_WORD[2][6] + 1;
    ARRAY_ARRAY_STRUCTURE_AUTO.ARRAY_ARRAY_WORD[2][7] := ARRAY_ARRAY_STRUCTURE_AUTO.ARRAY_ARRAY_WORD[2][7] + 1;
    ARRAY_ARRAY_STRUCTURE_AUTO.ARRAY_ARRAY_WORD[2][8] := ARRAY_ARRAY_STRUCTURE_AUTO.ARRAY_ARRAY_WORD[2][8] + 1;
    ARRAY_ARRAY_STRUCTURE_AUTO.ARRAY_ARRAY_WORD[2][9] := ARRAY_ARRAY_STRUCTURE_AUTO.ARRAY_ARRAY_WORD[2][9] + 1;

    ARRAY_ARRAY_STRUCTURE_AUTO.ARRAY_ARRAY_WORD[3][0] := ARRAY_ARRAY_STRUCTURE_AUTO.ARRAY_ARRAY_WORD[3][0] + 1;
    ARRAY_ARRAY_STRUCTURE_AUTO.ARRAY_ARRAY_WORD[3][1] := ARRAY_ARRAY_STRUCTURE_AUTO.ARRAY_ARRAY_WORD[3][1] + 1;
    ARRAY_ARRAY_STRUCTURE_AUTO.ARRAY_ARRAY_WORD[3][2] := ARRAY_ARRAY_STRUCTURE_AUTO.ARRAY_ARRAY_WORD[3][2] + 1;
    ARRAY_ARRAY_STRUCTURE_AUTO.ARRAY_ARRAY_WORD[3][3] := ARRAY_ARRAY_STRUCTURE_AUTO.ARRAY_ARRAY_WORD[3][3] + 1;
    ARRAY_ARRAY_STRUCTURE_AUTO.ARRAY_ARRAY_WORD[3][4] := ARRAY_ARRAY_STRUCTURE_AUTO.ARRAY_ARRAY_WORD[3][4] + 1;
    ARRAY_ARRAY_STRUCTURE_AUTO.ARRAY_ARRAY_WORD[3][5] := ARRAY_ARRAY_STRUCTURE_AUTO.ARRAY_ARRAY_WORD[3][5] + 1;
    ARRAY_ARRAY_STRUCTURE_AUTO.ARRAY_ARRAY_WORD[3][6] := ARRAY_ARRAY_STRUCTURE_AUTO.ARRAY_ARRAY_WORD[3][6] + 1;
    ARRAY_ARRAY_STRUCTURE_AUTO.ARRAY_ARRAY_WORD[3][7] := ARRAY_ARRAY_STRUCTURE_AUTO.ARRAY_ARRAY_WORD[3][7] + 1;
    ARRAY_ARRAY_STRUCTURE_AUTO.ARRAY_ARRAY_WORD[3][8] := ARRAY_ARRAY_STRUCTURE_AUTO.ARRAY_ARRAY_WORD[3][8] + 1;
    ARRAY_ARRAY_STRUCTURE_AUTO.ARRAY_ARRAY_WORD[3][9] := ARRAY_ARRAY_STRUCTURE_AUTO.ARRAY_ARRAY_WORD[3][9] + 1;

    ARRAY_ARRAY_STRUCTURE_AUTO.ARRAY_ARRAY_WORD[4][0] := ARRAY_ARRAY_STRUCTURE_AUTO.ARRAY_ARRAY_WORD[4][0] + 1;
    ARRAY_ARRAY_STRUCTURE_AUTO.ARRAY_ARRAY_WORD[4][1] := ARRAY_ARRAY_STRUCTURE_AUTO.ARRAY_ARRAY_WORD[4][1] + 1;
    ARRAY_ARRAY_STRUCTURE_AUTO.ARRAY_ARRAY_WORD[4][2] := ARRAY_ARRAY_STRUCTURE_AUTO.ARRAY_ARRAY_WORD[4][2] + 1;
    ARRAY_ARRAY_STRUCTURE_AUTO.ARRAY_ARRAY_WORD[4][3] := ARRAY_ARRAY_STRUCTURE_AUTO.ARRAY_ARRAY_WORD[4][3] + 1;
    ARRAY_ARRAY_STRUCTURE_AUTO.ARRAY_ARRAY_WORD[4][4] := ARRAY_ARRAY_STRUCTURE_AUTO.ARRAY_ARRAY_WORD[4][4] + 1;
    ARRAY_ARRAY_STRUCTURE_AUTO.ARRAY_ARRAY_WORD[4][5] := ARRAY_ARRAY_STRUCTURE_AUTO.ARRAY_ARRAY_WORD[4][5] + 1;
    ARRAY_ARRAY_STRUCTURE_AUTO.ARRAY_ARRAY_WORD[4][6] := ARRAY_ARRAY_STRUCTURE_AUTO.ARRAY_ARRAY_WORD[4][6] + 1;
    ARRAY_ARRAY_STRUCTURE_AUTO.ARRAY_ARRAY_WORD[4][7] := ARRAY_ARRAY_STRUCTURE_AUTO.ARRAY_ARRAY_WORD[4][7] + 1;
    ARRAY_ARRAY_STRUCTURE_AUTO.ARRAY_ARRAY_WORD[4][8] := ARRAY_ARRAY_STRUCTURE_AUTO.ARRAY_ARRAY_WORD[4][8] + 1;
    ARRAY_ARRAY_STRUCTURE_AUTO.ARRAY_ARRAY_WORD[4][9] := ARRAY_ARRAY_STRUCTURE_AUTO.ARRAY_ARRAY_WORD[4][9] + 1;

    ARRAY_ARRAY_STRUCTURE_AUTO.ARRAY_ARRAY_WORD[5][0] := ARRAY_ARRAY_STRUCTURE_AUTO.ARRAY_ARRAY_WORD[5][0] + 1;
    ARRAY_ARRAY_STRUCTURE_AUTO.ARRAY_ARRAY_WORD[5][1] := ARRAY_ARRAY_STRUCTURE_AUTO.ARRAY_ARRAY_WORD[5][1] + 1;
    ARRAY_ARRAY_STRUCTURE_AUTO.ARRAY_ARRAY_WORD[5][2] := ARRAY_ARRAY_STRUCTURE_AUTO.ARRAY_ARRAY_WORD[5][2] + 1;
    ARRAY_ARRAY_STRUCTURE_AUTO.ARRAY_ARRAY_WORD[5][3] := ARRAY_ARRAY_STRUCTURE_AUTO.ARRAY_ARRAY_WORD[5][3] + 1;
    ARRAY_ARRAY_STRUCTURE_AUTO.ARRAY_ARRAY_WORD[5][4] := ARRAY_ARRAY_STRUCTURE_AUTO.ARRAY_ARRAY_WORD[5][4] + 1;
    ARRAY_ARRAY_STRUCTURE_AUTO.ARRAY_ARRAY_WORD[5][5] := ARRAY_ARRAY_STRUCTURE_AUTO.ARRAY_ARRAY_WORD[5][5] + 1;
    ARRAY_ARRAY_STRUCTURE_AUTO.ARRAY_ARRAY_WORD[5][6] := ARRAY_ARRAY_STRUCTURE_AUTO.ARRAY_ARRAY_WORD[5][6] + 1;
    ARRAY_ARRAY_STRUCTURE_AUTO.ARRAY_ARRAY_WORD[5][7] := ARRAY_ARRAY_STRUCTURE_AUTO.ARRAY_ARRAY_WORD[5][7] + 1;
    ARRAY_ARRAY_STRUCTURE_AUTO.ARRAY_ARRAY_WORD[5][8] := ARRAY_ARRAY_STRUCTURE_AUTO.ARRAY_ARRAY_WORD[5][8] + 1;
    ARRAY_ARRAY_STRUCTURE_AUTO.ARRAY_ARRAY_WORD[5][9] := ARRAY_ARRAY_STRUCTURE_AUTO.ARRAY_ARRAY_WORD[5][9] + 1;

    ARRAY_ARRAY_STRUCTURE_AUTO.ARRAY_ARRAY_WORD[6][0] := ARRAY_ARRAY_STRUCTURE_AUTO.ARRAY_ARRAY_WORD[6][0] + 1;
    ARRAY_ARRAY_STRUCTURE_AUTO.ARRAY_ARRAY_WORD[6][1] := ARRAY_ARRAY_STRUCTURE_AUTO.ARRAY_ARRAY_WORD[6][1] + 1;
    ARRAY_ARRAY_STRUCTURE_AUTO.ARRAY_ARRAY_WORD[6][2] := ARRAY_ARRAY_STRUCTURE_AUTO.ARRAY_ARRAY_WORD[6][2] + 1;
    ARRAY_ARRAY_STRUCTURE_AUTO.ARRAY_ARRAY_WORD[6][3] := ARRAY_ARRAY_STRUCTURE_AUTO.ARRAY_ARRAY_WORD[6][3] + 1;
    ARRAY_ARRAY_STRUCTURE_AUTO.ARRAY_ARRAY_WORD[6][4] := ARRAY_ARRAY_STRUCTURE_AUTO.ARRAY_ARRAY_WORD[6][4] + 1;
    ARRAY_ARRAY_STRUCTURE_AUTO.ARRAY_ARRAY_WORD[6][5] := ARRAY_ARRAY_STRUCTURE_AUTO.ARRAY_ARRAY_WORD[6][5] + 1;
    ARRAY_ARRAY_STRUCTURE_AUTO.ARRAY_ARRAY_WORD[6][6] := ARRAY_ARRAY_STRUCTURE_AUTO.ARRAY_ARRAY_WORD[6][6] + 1;
    ARRAY_ARRAY_STRUCTURE_AUTO.ARRAY_ARRAY_WORD[6][7] := ARRAY_ARRAY_STRUCTURE_AUTO.ARRAY_ARRAY_WORD[6][7] + 1;
    ARRAY_ARRAY_STRUCTURE_AUTO.ARRAY_ARRAY_WORD[6][8] := ARRAY_ARRAY_STRUCTURE_AUTO.ARRAY_ARRAY_WORD[6][8] + 1;
    ARRAY_ARRAY_STRUCTURE_AUTO.ARRAY_ARRAY_WORD[6][9] := ARRAY_ARRAY_STRUCTURE_AUTO.ARRAY_ARRAY_WORD[6][9] + 1;

    ARRAY_ARRAY_STRUCTURE_AUTO.ARRAY_ARRAY_WORD[7][0] := ARRAY_ARRAY_STRUCTURE_AUTO.ARRAY_ARRAY_WORD[6][0];
    ARRAY_ARRAY_STRUCTURE_AUTO.ARRAY_ARRAY_WORD[7][1] := ARRAY_ARRAY_STRUCTURE_AUTO.ARRAY_ARRAY_WORD[6][1];
    ARRAY_ARRAY_STRUCTURE_AUTO.ARRAY_ARRAY_WORD[7][2] := ARRAY_ARRAY_STRUCTURE_AUTO.ARRAY_ARRAY_WORD[6][2];
    ARRAY_ARRAY_STRUCTURE_AUTO.ARRAY_ARRAY_WORD[7][3] := ARRAY_ARRAY_STRUCTURE_AUTO.ARRAY_ARRAY_WORD[6][3];
    ARRAY_ARRAY_STRUCTURE_AUTO.ARRAY_ARRAY_WORD[7][4] := ARRAY_ARRAY_STRUCTURE_AUTO.ARRAY_ARRAY_WORD[6][4];
    ARRAY_ARRAY_STRUCTURE_AUTO.ARRAY_ARRAY_WORD[7][5] := ARRAY_ARRAY_STRUCTURE_AUTO.ARRAY_ARRAY_WORD[6][5];
    ARRAY_ARRAY_STRUCTURE_AUTO.ARRAY_ARRAY_WORD[7][6] := ARRAY_ARRAY_STRUCTURE_AUTO.ARRAY_ARRAY_WORD[6][6];
    ARRAY_ARRAY_STRUCTURE_AUTO.ARRAY_ARRAY_WORD[7][7] := ARRAY_ARRAY_STRUCTURE_AUTO.ARRAY_ARRAY_WORD[6][7];
    ARRAY_ARRAY_STRUCTURE_AUTO.ARRAY_ARRAY_WORD[7][8] := ARRAY_ARRAY_STRUCTURE_AUTO.ARRAY_ARRAY_WORD[6][8];
    ARRAY_ARRAY_STRUCTURE_AUTO.ARRAY_ARRAY_WORD[7][9] := ARRAY_ARRAY_STRUCTURE_AUTO.ARRAY_ARRAY_WORD[6][9];

END_IF;

END_PROGRAM
